LIN {X 0,Y 303.722,Z 314.6,A -85,B 0,C 180,E1 -15936.643,E2 -15936.643} C_VEL
LIN {X 0,Y 304.019,Z 311.814,A -85,B 0,C 180,E1 -15938.642,E2 -15938.642} C_VEL
LIN {X 0,Y 304.561,Z 308.03,A -85,B 0,C 180,E1 -15940.638,E2 -15940.638} C_VEL
LIN {X 0,Y 305.432,Z 303.153,A -85,B 0,C 180,E1 -15942.626,E2 -15942.626} C_VEL
LIN {X 0,Y 306.814,Z 297.041,A -85,B 0,C 180,E1 -15944.594,E2 -15944.594} C_VEL
LIN {X 0,Y 308.414,Z 289.012,A -85,B 0,C 180,E1 -15946.664,E2 -15946.664} C_VEL
LIN {X 0,Y 310.224,Z 280.048,A -85,B 0,C 180,E1 -15948.491,E2 -15948.491} C_VEL
LIN {X 0,Y 312.464,Z 269.264,A -85,B 0,C 180,E1 -15950.231,E2 -15950.231} C_VEL
LIN {X 0,Y 314.317,Z 259.561,A -85,B 0,C 180,E1 -15951.477,E2 -15951.477} C_VEL
LIN {X 0,Y 316.058,Z 249.097,A -85,B 0,C 180,E1 -15952.555,E2 -15952.555} C_VEL
LIN {X 0,Y 317.837,Z 236.54,A -85,B 0,C 180,E1 -15953.54,E2 -15953.54} C_VEL
LIN {X 0,Y 319.26,Z 224.054,A -85,B 0,C 180,E1 -15954.247,E2 -15954.247} C_VEL
LIN {X 0,Y 320.237,Z 211.153,A -85,B 0,C 180,E1 -15954.73,E2 -15954.73} C_VEL
LIN {X 0,Y 321.791,Z 150.859,A -85,B 0,C 180,E1 -15956.133,E2 -15956.133} C_VEL
LIN {X 0,Y 318.654,Z 131.101,A -85,B 0,C 180,E1 -15956.979,E2 -15956.979} C_VEL
LIN {X 0,Y 314.024,Z 108.711,A -85,B 0,C 180,E1 -15958.092,E2 -15958.092} C_VEL
LIN {X 0,Y 312.285,Z 103.067,A -85,B 0,C 180,E1 -15958.447,E2 -15958.447} C_VEL
LIN {X 0,Y 310.254,Z 93.46,A -85,B 0,C 180,E1 -15961.399,E2 -15961.399} C_VEL
LIN {X 0,Y 308.062,Z 84.289,A -85,B 0,C 180,E1 -15964.395,E2 -15964.395} C_VEL
LIN {X 0,Y 305.495,Z 74.434,A -85,B 0,C 180,E1 -15967.849,E2 -15967.849} C_VEL
LIN {X 0,Y 305.439,Z 74.437,A -85,B 0,C 180,E1 -15971.856,E2 -15971.856} C_VEL
LIN {X 0,Y 305.408,Z 74.423,A -85,B 0,C 180,E1 -15975.509,E2 -15975.509} C_VEL
LIN {X 0,Y 305.473,Z 74.434,A -85,B 0,C 180,E1 -15978.149,E2 -15978.149} C_VEL
LIN {X 0,Y 305.506,Z 74.426,A -85,B 0,C 180,E1 -15981.602,E2 -15981.602} C_VEL
LIN {X 0,Y 305.46,Z 74.433,A -85,B 0,C 180,E1 -15984.887,E2 -15984.887} C_VEL
LIN {X 0,Y 305.45,Z 74.435,A -85,B 0,C 180,E1 -15988.354,E2 -15988.354} C_VEL
LIN {X 0,Y 305.518,Z 74.43,A -85,B 0,C 180,E1 -15991.114,E2 -15991.114} C_VEL
LIN {X 0,Y 305.569,Z 74.416,A -85,B 0,C 180,E1 -15994.088,E2 -15994.088} C_VEL
LIN {X 0,Y 305.501,Z 74.421,A -85,B 0,C 180,E1 -15998.403,E2 -15998.403} C_VEL
LIN {X 0,Y 305.589,Z 74.412,A -85,B 0,C 180,E1 -16001.218,E2 -16001.218} C_VEL
LIN {X 0,Y 305.646,Z 74.411,A -85,B 0,C 180,E1 -16005.349,E2 -16005.349} C_VEL
LIN {X 0,Y 305.636,Z 74.412,A -85,B 0,C 180,E1 -16009.4,E2 -16009.4} C_VEL
LIN {X 0,Y 305.805,Z 74.381,A -85,B 0,C 180,E1 -16012.074,E2 -16012.074} C_VEL
LIN {X 0,Y 305.684,Z 74.407,A -85,B 0,C 180,E1 -16014.724,E2 -16014.724} C_VEL
LIN {X 0,Y 305.955,Z 74.368,A -85,B 0,C 180,E1 -16018.684,E2 -16018.684} C_VEL
LIN {X 0,Y 305.953,Z 74.372,A -85,B 0,C 180,E1 -16021.317,E2 -16021.317} C_VEL
LIN {X 0,Y 305.68,Z 74.409,A -85,B 0,C 180,E1 -16025.277,E2 -16025.277} C_VEL
LIN {X 0,Y 305.769,Z 74.384,A -85,B 0,C 180,E1 -16027.927,E2 -16027.927} C_VEL
LIN {X 0,Y 305.597,Z 74.412,A -85,B 0,C 180,E1 -16031.946,E2 -16031.946} C_VEL
LIN {X 0,Y 305.607,Z 74.418,A -85,B 0,C 180,E1 -16035.015,E2 -16035.015} C_VEL
LIN {X 0,Y 305.542,Z 74.426,A -85,B 0,C 180,E1 -16039.428,E2 -16039.428} C_VEL
LIN {X 0,Y 305.484,Z 74.43,A -85,B 0,C 180,E1 -16043.04,E2 -16043.04} C_VEL
LIN {X 0,Y 305.476,Z 74.426,A -85,B 0,C 180,E1 -16046.201,E2 -16046.201} C_VEL
LIN {X 0,Y 305.461,Z 74.429,A -85,B 0,C 180,E1 -16049.039,E2 -16049.039} C_VEL
LIN {X 0,Y 305.436,Z 74.436,A -85,B 0,C 180,E1 -16051.954,E2 -16051.954} C_VEL
LIN {X 0,Y 305.461,Z 74.43,A -85,B 0,C 180,E1 -16055.114,E2 -16055.114} C_VEL
LIN {X 0,Y 305.434,Z 74.442,A -85,B 0,C 180,E1 -16058.526,E2 -16058.526} C_VEL
LIN {X 0,Y 305.426,Z 74.431,A -85,B 0,C 180,E1 -16061.86,E2 -16061.86} C_VEL
LIN {X 0,Y 305.411,Z 74.441,A -85,B 0,C 180,E1 -16065.938,E2 -16065.938} C_VEL
LIN {X 0,Y 305.48,Z 74.708,A -85,B 0,C 180,E1 -16066.355,E2 -16066.355} C_VEL
LIN {X 0,Y 305.822,Z 75.973,A -85,B 0,C 180,E1 -16066.792,E2 -16066.792} C_VEL
LIN {X 0,Y 313.965,Z 91.34,A -85,B 0,C 180,E1 -16068.219,E2 -16068.219} C_VEL
LIN {X 0,Y 321.333,Z 106.833,A -85,B 0,C 180,E1 -16069.468,E2 -16069.468} C_VEL
LIN {X 0,Y 323.152,Z 111.258,A -85,B 0,C 180,E1 -16069.78,E2 -16069.78} C_VEL
LIN {X 0,Y 320.986,Z 181.678,A -85,B 0,C 180,E1 -16071.391,E2 -16071.391} C_VEL
LIN {X 0,Y 320.123,Z 194.669,A -85,B 0,C 180,E1 -16071.92,E2 -16071.92} C_VEL
LIN {X 0,Y 319.072,Z 207.723,A -85,B 0,C 180,E1 -16072.738,E2 -16072.738} C_VEL
LIN {X 0,Y 317.642,Z 219.301,A -85,B 0,C 180,E1 -16073.712,E2 -16073.712} C_VEL
LIN {X 0,Y 315.904,Z 230.916,A -85,B 0,C 180,E1 -16074.989,E2 -16074.989} C_VEL
LIN {X 0,Y 314.114,Z 240.957,A -85,B 0,C 180,E1 -16076.375,E2 -16076.375} C_VEL
LIN {X 0,Y 312.149,Z 250.688,A -85,B 0,C 180,E1 -16078.056,E2 -16078.056} C_VEL
LIN {X 0,Y 310.584,Z 258.046,A -85,B 0,C 180,E1 -16079.627,E2 -16079.627} C_VEL
LIN {X 0,Y 308.977,Z 265.076,A -85,B 0,C 180,E1 -16081.468,E2 -16081.468} C_VEL
LIN {X 0,Y 307.432,Z 271.447,A -85,B 0,C 180,E1 -16083.564,E2 -16083.564} C_VEL
LIN {X 0,Y 306.27,Z 276.256,A -85,B 0,C 180,E1 -16085.604,E2 -16085.604} C_VEL
LIN {X 0,Y 305.351,Z 279.946,A -85,B 0,C 180,E1 -16087.681,E2 -16087.681} C_VEL
LIN {X 0,Y 304.641,Z 282.538,A -85,B 0,C 180,E1 -16089.755,E2 -16089.755} C_VEL
LIN {X 0,Y 304.213,Z 283.817,A -85,B 0,C 180,E1 -16091.298,E2 -16091.298} C_VEL
LIN {X 0,Y 303.812,Z 284.734,A -85,B 0,C 180,E1 -16093.884,E2 -16093.884} C_VEL
LIN {X 0,Y 303.721,Z 284.241,A -85,B 0,C 180,E1 -16096.379,E2 -16096.379} C_VEL
LIN {X 0,Y 303.759,Z 283.153,A -85,B 0,C 180,E1 -16097.982,E2 -16097.982} C_VEL
LIN {X 0,Y 303.804,Z 281.805,A -85,B 0,C 180,E1 -16099.335,E2 -16099.335} C_VEL
LIN {X 0,Y 304.108,Z 278.947,A -85,B 0,C 180,E1 -16101.361,E2 -16101.361} C_VEL
LIN {X 0,Y 304.502,Z 275.058,A -85,B 0,C 180,E1 -16103.374,E2 -16103.374} C_VEL
LIN {X 0,Y 304.981,Z 270.045,A -85,B 0,C 180,E1 -16105.374,E2 -16105.374} C_VEL
LIN {X 0,Y 305.676,Z 263.747,A -85,B 0,C 180,E1 -16107.365,E2 -16107.365} C_VEL
LIN {X 0,Y 306.671,Z 255.843,A -85,B 0,C 180,E1 -16109.344,E2 -16109.344} C_VEL
LIN {X 0,Y 307.685,Z 247.786,A -85,B 0,C 180,E1 -16110.982,E2 -16110.982} C_VEL
LIN {X 0,Y 308.861,Z 237.964,A -85,B 0,C 180,E1 -16112.609,E2 -16112.609} C_VEL
LIN {X 0,Y 310.052,Z 227.133,A -85,B 0,C 180,E1 -16114.044,E2 -16114.044} C_VEL
LIN {X 0,Y 311.02,Z 216.232,A -85,B 0,C 180,E1 -16115.186,E2 -16115.186} C_VEL
LIN {X 0,Y 311.857,Z 204.447,A -85,B 0,C 180,E1 -16116.146,E2 -16116.146} C_VEL
LIN {X 0,Y 312.535,Z 191.764,A -85,B 0,C 180,E1 -16116.902,E2 -16116.902} C_VEL
LIN {X 0,Y 313.021,Z 179.469,A -85,B 0,C 180,E1 -16117.378,E2 -16117.378} C_VEL
LIN {X 0,Y 314.626,Z 100.764,A -85,B 0,C 180,E1 -16119.182,E2 -16119.182} C_VEL
LIN {X 0,Y 309.281,Z 84.113,A -85,B 0,C 180,E1 -16119.931,E2 -16119.931} C_VEL
LIN {X 0,Y 305.662,Z 74.413,A -85,B 0,C 180,E1 -16120.435,E2 -16120.435} C_VEL
LIN {X 0,Y 305.643,Z 74.414,A -85,B 0,C 180,E1 -16125.035,E2 -16125.035} C_VEL
LIN {X 0,Y 305.58,Z 74.418,A -85,B 0,C 180,E1 -16129.445,E2 -16129.445} C_VEL
LIN {X 0,Y 305.49,Z 74.428,A -85,B 0,C 180,E1 -16133.039,E2 -16133.039} C_VEL
LIN {X 0,Y 305.536,Z 74.425,A -85,B 0,C 180,E1 -16136.221,E2 -16136.221} C_VEL
LIN {X 0,Y 305.492,Z 74.428,A -85,B 0,C 180,E1 -16139.047,E2 -16139.047} C_VEL
LIN {X 0,Y 305.447,Z 74.436,A -85,B 0,C 180,E1 -16141.952,E2 -16141.952} C_VEL
LIN {X 0,Y 305.467,Z 74.43,A -85,B 0,C 180,E1 -16145.113,E2 -16145.113} C_VEL
LIN {X 0,Y 305.472,Z 74.431,A -85,B 0,C 180,E1 -16148.533,E2 -16148.533} C_VEL
LIN {X 0,Y 305.481,Z 74.43,A -85,B 0,C 180,E1 -16152.59,E2 -16152.59} C_VEL
LIN {X 0,Y 305.447,Z 74.434,A -85,B 0,C 180,E1 -16156.348,E2 -16156.348} C_VEL
LIN {X 0,Y 305.449,Z 74.432,A -85,B 0,C 180,E1 -16160.05,E2 -16160.05} C_VEL
LIN {X 0,Y 304.746,Z 74.522,A -85,B 0,C 180,E1 -16161.151,E2 -16161.151} C_VEL
LIN {X 0,Y 301.917,Z 74.87,A -85,B 0,C 180,E1 -16162.945,E2 -16162.945} C_VEL
LIN {X 0,Y 299.531,Z 75.166,A -85,B 0,C 180,E1 -16164.4,E2 -16164.4} C_VEL
LIN {X 0,Y 298.487,Z 75.294,A -85,B 0,C 180,E1 -16165.525,E2 -16165.525} C_VEL
LIN {X 0,Y 298.39,Z 75.305,A -85,B 0,C 180,E1 -16165.907,E2 -16165.907} C_VEL
LIN {X 0,Y 298.395,Z 75.314,A -85,B 0,C 180,E1 -16168.791,E2 -16168.791} C_VEL
LIN {X 0,Y 298.46,Z 75.305,A -85,B 0,C 180,E1 -16171.903,E2 -16171.903} C_VEL
LIN {X 0,Y 298.486,Z 75.301,A -85,B 0,C 180,E1 -16174.924,E2 -16174.924} C_VEL
LIN {X 0,Y 298.454,Z 75.306,A -85,B 0,C 180,E1 -16179.315,E2 -16179.315} C_VEL
LIN {X 0,Y 298.541,Z 75.297,A -85,B 0,C 180,E1 -16182.179,E2 -16182.179} C_VEL
LIN {X 0,Y 298.596,Z 75.287,A -85,B 0,C 180,E1 -16184.995,E2 -16184.995} C_VEL
LIN {X 0,Y 298.594,Z 75.288,A -85,B 0,C 180,E1 -16189.146,E2 -16189.146} C_VEL
LIN {X 0,Y 298.744,Z 75.27,A -85,B 0,C 180,E1 -16191.885,E2 -16191.885} C_VEL
LIN {X 0,Y 298.658,Z 75.28,A -85,B 0,C 180,E1 -16194.599,E2 -16194.599} C_VEL
LIN {X 0,Y 298.924,Z 75.245,A -85,B 0,C 180,E1 -16198.652,E2 -16198.652} C_VEL
LIN {X 0,Y 298.924,Z 75.246,A -85,B 0,C 180,E1 -16201.347,E2 -16201.347} C_VEL
LIN {X 0,Y 298.778,Z 75.264,A -85,B 0,C 180,E1 -16206.754,E2 -16206.754} C_VEL
LIN {X 0,Y 298.628,Z 75.287,A -85,B 0,C 180,E1 -16209.482,E2 -16209.482} C_VEL
LIN {X 0,Y 298.555,Z 75.294,A -85,B 0,C 180,E1 -16213.615,E2 -16213.615} C_VEL
LIN {X 0,Y 298.551,Z 75.292,A -85,B 0,C 180,E1 -16216.408,E2 -16216.408} C_VEL
LIN {X 0,Y 298.512,Z 75.299,A -85,B 0,C 180,E1 -16219.653,E2 -16219.653} C_VEL
LIN {X 0,Y 298.43,Z 75.309,A -85,B 0,C 180,E1 -16223.6,E2 -16223.6} C_VEL
LIN {X 0,Y 298.487,Z 75.303,A -85,B 0,C 180,E1 -16226.574,E2 -16226.574} C_VEL
LIN {X 0,Y 298.423,Z 75.307,A -85,B 0,C 180,E1 -16229.641,E2 -16229.641} C_VEL
LIN {X 0,Y 298.397,Z 75.316,A -85,B 0,C 180,E1 -16232.8,E2 -16232.8} C_VEL
LIN {X 0,Y 298.448,Z 75.309,A -85,B 0,C 180,E1 -16236.807,E2 -16236.807} C_VEL
LIN {X 0,Y 298.388,Z 75.315,A -85,B 0,C 180,E1 -16241.087,E2 -16241.087} C_VEL
LIN {X 0,Y 298.4,Z 75.312,A -85,B 0,C 180,E1 -16243.103,E2 -16243.103} C_VEL
LIN {X 0,Y 298.404,Z 75.313,A -85,B 0,C 180,E1 -16246.92,E2 -16246.92} C_VEL
LIN {X 0,Y 298.416,Z 75.312,A -85,B 0,C 180,E1 -16251.003,E2 -16251.003} C_VEL
LIN {X 0,Y 298.433,Z 75.314,A -85,B 0,C 180,E1 -16253.932,E2 -16253.932} C_VEL
LIN {X 0,Y 298.456,Z 75.334,A -85,B 0,C 180,E1 -16257.363,E2 -16257.363} C_VEL
LIN {X 0,Y 301.125,Z 88.007,A -85,B 0,C 180,E1 -16261.034,E2 -16261.034} C_VEL
LIN {X 0,Y 302.351,Z 95.258,A -85,B 0,C 180,E1 -16263.046,E2 -16263.046} C_VEL
LIN {X 0,Y 301.429,Z 103.913,A -85,B 0,C 180,E1 -16265.263,E2 -16265.263} C_VEL
LIN {X 0,Y 306.811,Z 147.996,A -85,B 0,C 180,E1 -16266.715,E2 -16266.715} C_VEL
LIN {X 0,Y 306.88,Z 159.405,A -85,B 0,C 180,E1 -16266.998,E2 -16266.998} C_VEL
LIN {X 0,Y 305.694,Z 213.727,A -85,B 0,C 180,E1 -16268.296,E2 -16268.296} C_VEL
LIN {X 0,Y 304.904,Z 227.31,A -85,B 0,C 180,E1 -16268.89,E2 -16268.89} C_VEL
LIN {X 0,Y 303.903,Z 239.769,A -85,B 0,C 180,E1 -16269.702,E2 -16269.702} C_VEL
LIN {X 0,Y 302.735,Z 250.891,A -85,B 0,C 180,E1 -16270.681,E2 -16270.681} C_VEL
LIN {X 0,Y 301.478,Z 261.198,A -85,B 0,C 180,E1 -16271.832,E2 -16271.832} C_VEL
LIN {X 0,Y 300.34,Z 271.925,A -85,B 0,C 180,E1 -16273.342,E2 -16273.342} C_VEL
LIN {X 0,Y 299.397,Z 280.34,A -85,B 0,C 180,E1 -16274.797,E2 -16274.797} C_VEL
LIN {X 0,Y 298.329,Z 289.451,A -85,B 0,C 180,E1 -16276.721,E2 -16276.721} C_VEL
LIN {X 0,Y 297.404,Z 297.125,A -85,B 0,C 180,E1 -16278.757,E2 -16278.757} C_VEL
LIN {X 0,Y 296.926,Z 304.228,A -85,B 0,C 180,E1 -16281.149,E2 -16281.149} C_VEL
LIN {X 0,Y 296.685,Z 308.907,A -85,B 0,C 180,E1 -16283.197,E2 -16283.197} C_VEL
LIN {X 0,Y 296.635,Z 312.451,A -85,B 0,C 180,E1 -16285.243,E2 -16285.243} C_VEL
LIN {X 0,Y 296.692,Z 314.96,A -85,B 0,C 180,E1 -16287.284,E2 -16287.284} C_VEL
LIN {X 0,Y 296.771,Z 316.11,A -85,B 0,C 180,E1 -16288.643,E2 -16288.643} C_VEL
LIN {X 0,Y 296.857,Z 316.815,A -85,B 0,C 180,E1 -16290,E2 -16290} C_VEL
LIN {X 0,Y 296.623,Z 317.027,A -85,B 0,C 180,E1 -16292.716,E2 -16292.716} C_VEL
LIN {X 0,Y 296.596,Z 316.546,A -85,B 0,C 180,E1 -16294.076,E2 -16294.076} C_VEL
LIN {X 0,Y 296.644,Z 314.324,A -85,B 0,C 180,E1 -16296.803,E2 -16296.803} C_VEL
LIN {X 0,Y 296.975,Z 311.593,A -85,B 0,C 180,E1 -16298.848,E2 -16298.848} C_VEL
LIN {X 0,Y 297.544,Z 307.864,A -85,B 0,C 180,E1 -16300.892,E2 -16300.892} C_VEL
LIN {X 0,Y 298.487,Z 303.048,A -85,B 0,C 180,E1 -16302.925,E2 -16302.925} C_VEL
LIN {X 0,Y 300.18,Z 295.88,A -85,B 0,C 180,E1 -16305.271,E2 -16305.271} C_VEL
LIN {X 0,Y 301.737,Z 288.176,A -85,B 0,C 180,E1 -16307.261,E2 -16307.261} C_VEL
LIN {X 0,Y 303.918,Z 278.435,A -85,B 0,C 180,E1 -16309.239,E2 -16309.239} C_VEL
LIN {X 0,Y 306.043,Z 268.475,A -85,B 0,C 180,E1 -16310.851,E2 -16310.851} C_VEL
LIN {X 0,Y 308.045,Z 258.665,A -85,B 0,C 180,E1 -16312.113,E2 -16312.113} C_VEL
LIN {X 0,Y 309.834,Z 248.056,A -85,B 0,C 180,E1 -16313.21,E2 -16313.21} C_VEL
LIN {X 0,Y 311.716,Z 235.322,A -85,B 0,C 180,E1 -16314.208,E2 -16314.208} C_VEL
LIN {X 0,Y 313.192,Z 222.536,A -85,B 0,C 180,E1 -16314.926,E2 -16314.926} C_VEL
LIN {X 0,Y 314.069,Z 209.411,A -85,B 0,C 180,E1 -16315.405,E2 -16315.405} C_VEL
LIN {X 0,Y 315.77,Z 152.738,A -85,B 0,C 180,E1 -16316.726,E2 -16316.726} C_VEL
LIN {X 0,Y 312.775,Z 133.284,A -85,B 0,C 180,E1 -16317.577,E2 -16317.577} C_VEL
LIN {X 0,Y 308.218,Z 110.954,A -85,B 0,C 180,E1 -16318.718,E2 -16318.718} C_VEL
LIN {X 0,Y 306.786,Z 106.516,A -85,B 0,C 180,E1 -16319.016,E2 -16319.016} C_VEL
LIN {X 0,Y 305.043,Z 102.497,A -85,B 0,C 180,E1 -16319.37,E2 -16319.37} C_VEL
LIN {X 0,Y 302.639,Z 91.519,A -85,B 0,C 180,E1 -16322.9,E2 -16322.9} C_VEL
LIN {X 0,Y 299.836,Z 80.463,A -85,B 0,C 180,E1 -16326.743,E2 -16326.743} C_VEL
LIN {X 0,Y 298.421,Z 75.312,A -85,B 0,C 180,E1 -16328.681,E2 -16328.681} C_VEL
LIN {X 0,Y 298.397,Z 75.317,A -85,B 0,C 180,E1 -16333.103,E2 -16333.103} C_VEL
LIN {X 0,Y 298.43,Z 75.302,A -85,B 0,C 180,E1 -16336.926,E2 -16336.926} C_VEL
LIN {X 0,Y 298.424,Z 75.313,A -85,B 0,C 180,E1 -16341.001,E2 -16341.001} C_VEL
LIN {X 0,Y 298.43,Z 75.311,A -85,B 0,C 180,E1 -16343.932,E2 -16343.932} C_VEL
LIN {X 0,Y 298.393,Z 75.315,A -85,B 0,C 180,E1 -16347.983,E2 -16347.983} C_VEL
LIN {X 0,Y 298.461,Z 75.306,A -85,B 0,C 180,E1 -16351.904,E2 -16351.904} C_VEL
LIN {X 0,Y 298.483,Z 75.305,A -85,B 0,C 180,E1 -16354.924,E2 -16354.924} C_VEL
LIN {X 0,Y 298.454,Z 75.307,A -85,B 0,C 180,E1 -16359.316,E2 -16359.316} C_VEL
LIN {X 0,Y 298.536,Z 75.286,A -85,B 0,C 180,E1 -16362.179,E2 -16362.179} C_VEL
LIN {X 0,Y 298.591,Z 75.29,A -85,B 0,C 180,E1 -16364.995,E2 -16364.995} C_VEL
LIN {X 0,Y 298.591,Z 75.29,A -85,B 0,C 180,E1 -16369.147,E2 -16369.147} C_VEL
LIN {X 0,Y 298.752,Z 75.26,A -85,B 0,C 180,E1 -16371.886,E2 -16371.886} C_VEL
LIN {X 0,Y 298.655,Z 75.283,A -85,B 0,C 180,E1 -16374.599,E2 -16374.599} C_VEL
LIN {X 0,Y 298.921,Z 75.243,A -85,B 0,C 180,E1 -16378.653,E2 -16378.653} C_VEL
LIN {X 0,Y 298.919,Z 75.247,A -85,B 0,C 180,E1 -16381.348,E2 -16381.348} C_VEL
LIN {X 0,Y 298.773,Z 75.265,A -85,B 0,C 180,E1 -16386.755,E2 -16386.755} C_VEL
LIN {X 0,Y 298.623,Z 75.282,A -85,B 0,C 180,E1 -16389.483,E2 -16389.483} C_VEL
LIN {X 0,Y 298.543,Z 75.288,A -85,B 0,C 180,E1 -16393.616,E2 -16393.616} C_VEL
LIN {X 0,Y 298.485,Z 75.302,A -85,B 0,C 180,E1 -16396.413,E2 -16396.413} C_VEL
LIN {X 0,Y 298.482,Z 75.305,A -85,B 0,C 180,E1 -16399.64,E2 -16399.64} C_VEL
LIN {X 0,Y 298.423,Z 75.312,A -85,B 0,C 180,E1 -16403.601,E2 -16403.601} C_VEL
LIN {X 0,Y 298.415,Z 75.308,A -85,B 0,C 180,E1 -16406.582,E2 -16406.582} C_VEL
LIN {X 0,Y 298.399,Z 75.309,A -85,B 0,C 180,E1 -16409.644,E2 -16409.644} C_VEL
LIN {X 0,Y 298.392,Z 75.312,A -85,B 0,C 180,E1 -16412.801,E2 -16412.801} C_VEL
LIN {X 0,Y 298.441,Z 75.312,A -85,B 0,C 180,E1 -16416.807,E2 -16416.807} C_VEL
LIN {X 0,Y 298.38,Z 75.306,A -85,B 0,C 180,E1 -16421.087,E2 -16421.087} C_VEL
LIN {X 0,Y 298.399,Z 75.324,A -85,B 0,C 180,E1 -16423.104,E2 -16423.104} C_VEL
LIN {X 0,Y 298.375,Z 75.401,A -85,B 0,C 180,E1 -16425.5,E2 -16425.5} C_VEL
LIN {X 0,Y 298.533,Z 76.217,A -85,B 0,C 180,E1 -16425.831,E2 -16425.831} C_VEL
LIN {X 0,Y 300.086,Z 79.172,A -85,B 0,C 180,E1 -16426.129,E2 -16426.129} C_VEL
LIN {X 0,Y 307.562,Z 92.858,A -85,B 0,C 180,E1 -16427.486,E2 -16427.486} C_VEL
LIN {X 0,Y 315.028,Z 108.392,A -85,B 0,C 180,E1 -16428.8,E2 -16428.8} C_VEL
LIN {X 0,Y 317.041,Z 113.075,A -85,B 0,C 180,E1 -16429.154,E2 -16429.154} C_VEL
LIN {X 0,Y 314.826,Z 182.102,A -85,B 0,C 180,E1 -16430.762,E2 -16430.762} C_VEL
LIN {X 0,Y 313.876,Z 195.801,A -85,B 0,C 180,E1 -16431.338,E2 -16431.338} C_VEL
LIN {X 0,Y 312.81,Z 208.298,A -85,B 0,C 180,E1 -16432.144,E2 -16432.144} C_VEL
LIN {X 0,Y 311.415,Z 219.156,A -85,B 0,C 180,E1 -16433.068,E2 -16433.068} C_VEL
LIN {X 0,Y 309.73,Z 229.943,A -85,B 0,C 180,E1 -16434.249,E2 -16434.249} C_VEL
LIN {X 0,Y 307.726,Z 240.977,A -85,B 0,C 180,E1 -16435.779,E2 -16435.779} C_VEL
LIN {X 0,Y 305.818,Z 249.892,A -85,B 0,C 180,E1 -16437.313,E2 -16437.313} C_VEL
LIN {X 0,Y 303.966,Z 258.346,A -85,B 0,C 180,E1 -16439.128,E2 -16439.128} C_VEL
LIN {X 0,Y 302.147,Z 265.846,A -85,B 0,C 180,E1 -16441.142,E2 -16441.142} C_VEL
LIN {X 0,Y 300.677,Z 271.54,A -85,B 0,C 180,E1 -16443.055,E2 -16443.055} C_VEL
LIN {X 0,Y 299.487,Z 276.156,A -85,B 0,C 180,E1 -16445.014,E2 -16445.014} C_VEL
LIN {X 0,Y 298.725,Z 279.091,A -85,B 0,C 180,E1 -16446.57,E2 -16446.57} C_VEL
LIN {X 0,Y 298.212,Z 281.006,A -85,B 0,C 180,E1 -16447.848,E2 -16447.848} C_VEL
LIN {X 0,Y 297.714,Z 282.682,A -85,B 0,C 180,E1 -16449.262,E2 -16449.262} C_VEL
LIN {X 0,Y 297.201,Z 284.199,A -85,B 0,C 180,E1 -16451.068,E2 -16451.068} C_VEL
LIN {X 0,Y 296.761,Z 285.1,A -85,B 0,C 180,E1 -16453.49,E2 -16453.49} C_VEL
LIN {X 0,Y 296.635,Z 284.634,A -85,B 0,C 180,E1 -16456.264,E2 -16456.264} C_VEL
LIN {X 0,Y 296.651,Z 283.735,A -85,B 0,C 180,E1 -16457.689,E2 -16457.689} C_VEL
LIN {X 0,Y 296.691,Z 282.44,A -85,B 0,C 180,E1 -16459.077,E2 -16459.077} C_VEL
LIN {X 0,Y 296.982,Z 279.693,A -85,B 0,C 180,E1 -16461.152,E2 -16461.152} C_VEL
LIN {X 0,Y 297.391,Z 275.921,A -85,B 0,C 180,E1 -16463.215,E2 -16463.215} C_VEL
LIN {X 0,Y 297.857,Z 271.035,A -85,B 0,C 180,E1 -16465.263,E2 -16465.263} C_VEL
LIN {X 0,Y 298.564,Z 264.877,A -85,B 0,C 180,E1 -16467.302,E2 -16467.302} C_VEL
LIN {X 0,Y 299.561,Z 257.21,A -85,B 0,C 180,E1 -16469.328,E2 -16469.328} C_VEL
LIN {X 0,Y 300.582,Z 249.354,A -85,B 0,C 180,E1 -16471.005,E2 -16471.005} C_VEL
LIN {X 0,Y 301.764,Z 239.77,A -85,B 0,C 180,E1 -16472.67,E2 -16472.67} C_VEL
LIN {X 0,Y 303.023,Z 228.766,A -85,B 0,C 180,E1 -16474.204,E2 -16474.204} C_VEL
LIN {X 0,Y 304.13,Z 217.193,A -85,B 0,C 180,E1 -16475.47,E2 -16475.47} C_VEL
LIN {X 0,Y 305.065,Z 204.451,A -85,B 0,C 180,E1 -16476.532,E2 -16476.532} C_VEL
LIN {X 0,Y 305.773,Z 191.588,A -85,B 0,C 180,E1 -16477.304,E2 -16477.304} C_VEL
LIN {X 0,Y 306.27,Z 178.865,A -85,B 0,C 180,E1 -16477.79,E2 -16477.79} C_VEL
LIN {X 0,Y 307.887,Z 101.929,A -85,B 0,C 180,E1 -16479.587,E2 -16479.587} C_VEL
LIN {X 0,Y 302.49,Z 85.456,A -85,B 0,C 180,E1 -16480.359,E2 -16480.359} C_VEL
LIN {X 0,Y 298.69,Z 75.916,A -85,B 0,C 180,E1 -16480.869,E2 -16480.869} C_VEL
LIN {X 0,Y 298.577,Z 75.296,A -85,B 0,C 180,E1 -16480.94,E2 -16480.94} C_VEL
LIN {X 0,Y 298.61,Z 75.29,A -85,B 0,C 180,E1 -16485.209,E2 -16485.209} C_VEL
LIN {X 0,Y 298.543,Z 75.294,A -85,B 0,C 180,E1 -16489.243,E2 -16489.243} C_VEL
LIN {X 0,Y 298.433,Z 75.309,A -85,B 0,C 180,E1 -16493.6,E2 -16493.6} C_VEL
LIN {X 0,Y 298.491,Z 75.3,A -85,B 0,C 180,E1 -16496.575,E2 -16496.575} C_VEL
LIN {X 0,Y 298.421,Z 75.312,A -85,B 0,C 180,E1 -16499.641,E2 -16499.641} C_VEL
LIN {X 0,Y 298.4,Z 75.31,A -85,B 0,C 180,E1 -16502.8,E2 -16502.8} C_VEL
LIN {X 0,Y 298.469,Z 75.304,A -85,B 0,C 180,E1 -16506.812,E2 -16506.812} C_VEL
LIN {X 0,Y 298.416,Z 75.311,A -85,B 0,C 180,E1 -16511.093,E2 -16511.093} C_VEL
LIN {X 0,Y 298.43,Z 75.311,A -85,B 0,C 180,E1 -16513.109,E2 -16513.109} C_VEL
LIN {X 0,Y 298.406,Z 75.312,A -85,B 0,C 180,E1 -16516.921,E2 -16516.921} C_VEL
LIN {X 0,Y 298.402,Z 75.313,A -85,B 0,C 180,E1 -16521.007,E2 -16521.007} C_VEL
LIN {X 0,Y 298.421,Z 75.298,A -85,B 0,C 180,E1 -16523.93,E2 -16523.93} C_VEL
LIN {X 0,Y 298.39,Z 75.305,A -85,B 0,C 180,E1 -16525.907,E2 -16525.907} C_VEL
LIN {X 0,Y 297.689,Z 75.398,A -85,B 0,C 180,E1 -16527.034,E2 -16527.034} C_VEL
LIN {X 0,Y 294.834,Z 75.758,A -85,B 0,C 180,E1 -16528.869,E2 -16528.869} C_VEL
LIN {X 0,Y 292.448,Z 76.055,A -85,B 0,C 180,E1 -16530.359,E2 -16530.359} C_VEL
LIN {X 0,Y 291.445,Z 76.18,A -85,B 0,C 180,E1 -16531.513,E2 -16531.513} C_VEL
LIN {X 0,Y 291.373,Z 76.188,A -85,B 0,C 180,E1 -16531.903,E2 -16531.903} C_VEL
LIN {X 0,Y 291.416,Z 76.183,A -85,B 0,C 180,E1 -16534.271,E2 -16534.271} C_VEL
LIN {X 0,Y 291.385,Z 76.186,A -85,B 0,C 180,E1 -16537.299,E2 -16537.299} C_VEL
LIN {X 0,Y 291.461,Z 76.18,A -85,B 0,C 180,E1 -16540.27,E2 -16540.27} C_VEL
LIN {X 0,Y 291.558,Z 76.165,A -85,B 0,C 180,E1 -16544.623,E2 -16544.623} C_VEL
LIN {X 0,Y 291.538,Z 76.167,A -85,B 0,C 180,E1 -16548.88,E2 -16548.88} C_VEL
LIN {X 0,Y 291.691,Z 76.147,A -85,B 0,C 180,E1 -16551.688,E2 -16551.688} C_VEL
LIN {X 0,Y 291.629,Z 76.157,A -85,B 0,C 180,E1 -16554.468,E2 -16554.468} C_VEL
LIN {X 0,Y 291.891,Z 76.121,A -85,B 0,C 180,E1 -16558.62,E2 -16558.62} C_VEL
LIN {X 0,Y 291.891,Z 76.122,A -85,B 0,C 180,E1 -16561.379,E2 -16561.379} C_VEL
LIN {X 0,Y 291.725,Z 76.143,A -85,B 0,C 180,E1 -16566.918,E2 -16566.918} C_VEL
LIN {X 0,Y 291.57,Z 76.165,A -85,B 0,C 180,E1 -16569.714,E2 -16569.714} C_VEL
LIN {X 0,Y 291.524,Z 76.168,A -85,B 0,C 180,E1 -16573.95,E2 -16573.95} C_VEL
LIN {X 0,Y 291.489,Z 76.173,A -85,B 0,C 180,E1 -16576.817,E2 -16576.817} C_VEL
LIN {X 0,Y 291.453,Z 76.178,A -85,B 0,C 180,E1 -16579.874,E2 -16579.874} C_VEL
LIN {X 0,Y 291.384,Z 76.187,A -85,B 0,C 180,E1 -16584.207,E2 -16584.207} C_VEL
LIN {X 0,Y 291.422,Z 76.183,A -85,B 0,C 180,E1 -16587.271,E2 -16587.271} C_VEL
LIN {X 0,Y 291.339,Z 76.192,A -85,B 0,C 180,E1 -16590.436,E2 -16590.436} C_VEL
LIN {X 0,Y 291.347,Z 76.191,A -85,B 0,C 180,E1 -16593.698,E2 -16593.698} C_VEL
LIN {X 0,Y 291.377,Z 76.188,A -85,B 0,C 180,E1 -16597.254,E2 -16597.254} C_VEL
LIN {X 0,Y 291.334,Z 76.196,A -85,B 0,C 180,E1 -16600.642,E2 -16600.642} C_VEL
LIN {X 0,Y 291.292,Z 76.197,A -85,B 0,C 180,E1 -16604.402,E2 -16604.402} C_VEL
LIN {X 0,Y 291.328,Z 76.197,A -85,B 0,C 180,E1 -16608.404,E2 -16608.404} C_VEL
LIN {X 0,Y 291.366,Z 76.191,A -85,B 0,C 180,E1 -16611.16,E2 -16611.16} C_VEL
LIN {X 0,Y 291.387,Z 76.189,A -85,B 0,C 180,E1 -16614.629,E2 -16614.629} C_VEL
LIN {X 0,Y 291.415,Z 76.335,A -85,B 0,C 180,E1 -16617.027,E2 -16617.027} C_VEL
LIN {X 0,Y 293.998,Z 88.511,A -85,B 0,C 180,E1 -16620.656,E2 -16620.656} C_VEL
LIN {X 0,Y 295.32,Z 95.896,A -85,B 0,C 180,E1 -16622.766,E2 -16622.766} C_VEL
LIN {X 0,Y 294.691,Z 102.77,A -85,B 0,C 180,E1 -16624.578,E2 -16624.578} C_VEL
LIN {X 0,Y 294.606,Z 103.493,A -85,B 0,C 180,E1 -16624.767,E2 -16624.767} C_VEL
LIN {X 0,Y 299.795,Z 146.157,A -85,B 0,C 180,E1 -16626.222,E2 -16626.222} C_VEL
LIN {X 0,Y 300.277,Z 151.887,A -85,B 0,C 180,E1 -16626.397,E2 -16626.397} C_VEL
LIN {X 0,Y 298.948,Z 212.642,A -85,B 0,C 180,E1 -16627.867,E2 -16627.867} C_VEL
LIN {X 0,Y 298.218,Z 225.762,A -85,B 0,C 180,E1 -16628.439,E2 -16628.439} C_VEL
LIN {X 0,Y 297.22,Z 237.983,A -85,B 0,C 180,E1 -16629.225,E2 -16629.225} C_VEL
LIN {X 0,Y 296.045,Z 249.496,A -85,B 0,C 180,E1 -16630.227,E2 -16630.227} C_VEL
LIN {X 0,Y 294.528,Z 261.296,A -85,B 0,C 180,E1 -16631.568,E2 -16631.568} C_VEL
LIN {X 0,Y 293.358,Z 271.941,A -85,B 0,C 180,E1 -16633.113,E2 -16633.113} C_VEL
LIN {X 0,Y 292.447,Z 279.164,A -85,B 0,C 180,E1 -16634.385,E2 -16634.385} C_VEL
LIN {X 0,Y 291.353,Z 288.611,A -85,B 0,C 180,E1 -16636.397,E2 -16636.397} C_VEL
LIN {X 0,Y 290.401,Z 296.384,A -85,B 0,C 180,E1 -16638.483,E2 -16638.483} C_VEL
LIN {X 0,Y 289.994,Z 301.712,A -85,B 0,C 180,E1 -16640.232,E2 -16640.232} C_VEL
LIN {X 0,Y 289.689,Z 306.852,A -85,B 0,C 180,E1 -16642.332,E2 -16642.332} C_VEL
LIN {X 0,Y 289.542,Z 311.507,A -85,B 0,C 180,E1 -16644.873,E2 -16644.873} C_VEL
LIN {X 0,Y 289.613,Z 314.461,A -85,B 0,C 180,E1 -16647.218,E2 -16647.218} C_VEL
LIN {X 0,Y 289.678,Z 315.652,A -85,B 0,C 180,E1 -16648.609,E2 -16648.609} C_VEL
LIN {X 0,Y 289.767,Z 316.392,A -85,B 0,C 180,E1 -16649.999,E2 -16649.999} C_VEL
LIN {X 0,Y 289.544,Z 316.654,A -85,B 0,C 180,E1 -16652.782,E2 -16652.782} C_VEL
LIN {X 0,Y 289.509,Z 316.206,A -85,B 0,C 180,E1 -16654.176,E2 -16654.176} C_VEL
LIN {X 0,Y 289.48,Z 315.332,A -85,B 0,C 180,E1 -16655.572,E2 -16655.572} C_VEL
LIN {X 0,Y 289.772,Z 312.371,A -85,B 0,C 180,E1 -16658.367,E2 -16658.367} C_VEL
LIN {X 0,Y 290.302,Z 309.032,A -85,B 0,C 180,E1 -16660.461,E2 -16660.461} C_VEL
LIN {X 0,Y 291.115,Z 304.647,A -85,B 0,C 180,E1 -16662.548,E2 -16662.548} C_VEL
LIN {X 0,Y 292.805,Z 298.079,A -85,B 0,C 180,E1 -16664.952,E2 -16664.952} C_VEL
LIN {X 0,Y 294.351,Z 291.194,A -85,B 0,C 180,E1 -16666.931,E2 -16666.931} C_VEL
LIN {X 0,Y 296.028,Z 283.668,A -85,B 0,C 180,E1 -16668.693,E2 -16668.693} C_VEL
LIN {X 0,Y 298.079,Z 274.925,A -85,B 0,C 180,E1 -16670.35,E2 -16670.35} C_VEL
LIN {X 0,Y 300.364,Z 264.202,A -85,B 0,C 180,E1 -16671.985,E2 -16671.985} C_VEL
LIN {X 0,Y 302.469,Z 253.528,A -85,B 0,C 180,E1 -16673.265,E2 -16673.265} C_VEL
LIN {X 0,Y 304.52,Z 241.587,A -85,B 0,C 180,E1 -16674.364,E2 -16674.364} C_VEL
LIN {X 0,Y 306.207,Z 229.196,A -85,B 0,C 180,E1 -16675.216,E2 -16675.216} C_VEL
LIN {X 0,Y 307.533,Z 215.935,A -85,B 0,C 180,E1 -16675.844,E2 -16675.844} C_VEL
LIN {X 0,Y 308.293,Z 199.707,A -85,B 0,C 180,E1 -16676.296,E2 -16676.296} C_VEL
LIN {X 0,Y 309.639,Z 153.176,A -85,B 0,C 180,E1 -16677.399,E2 -16677.399} C_VEL
LIN {X 0,Y 306.449,Z 132.847,A -85,B 0,C 180,E1 -16678.328,E2 -16678.328} C_VEL
LIN {X 0,Y 302.217,Z 112.29,A -85,B 0,C 180,E1 -16679.427,E2 -16679.427} C_VEL
LIN {X 0,Y 299.224,Z 105.508,A -85,B 0,C 180,E1 -16680.009,E2 -16680.009} C_VEL
LIN {X 0,Y 297.776,Z 101.976,A -85,B 0,C 180,E1 -16680.335,E2 -16680.335} C_VEL
LIN {X 0,Y 295.243,Z 90.716,A -85,B 0,C 180,E1 -16684.121,E2 -16684.121} C_VEL
LIN {X 0,Y 292.743,Z 81.145,A -85,B 0,C 180,E1 -16687.604,E2 -16687.604} C_VEL
LIN {X 0,Y 291.369,Z 76.192,A -85,B 0,C 180,E1 -16689.6,E2 -16689.6} C_VEL
LIN {X 0,Y 291.307,Z 76.198,A -85,B 0,C 180,E1 -16693.633,E2 -16693.633} C_VEL
LIN {X 0,Y 291.349,Z 76.191,A -85,B 0,C 180,E1 -16697.513,E2 -16697.513} C_VEL
LIN {X 0,Y 291.373,Z 76.191,A -85,B 0,C 180,E1 -16701.162,E2 -16701.162} C_VEL
LIN {X 0,Y 291.383,Z 76.188,A -85,B 0,C 180,E1 -16704.629,E2 -16704.629} C_VEL
LIN {X 0,Y 291.37,Z 76.19,A -85,B 0,C 180,E1 -16707.951,E2 -16707.951} C_VEL
LIN {X 0,Y 291.38,Z 76.191,A -85,B 0,C 180,E1 -16711.158,E2 -16711.158} C_VEL
LIN {X 0,Y 291.414,Z 76.179,A -85,B 0,C 180,E1 -16714.272,E2 -16714.272} C_VEL
LIN {X 0,Y 291.38,Z 76.177,A -85,B 0,C 180,E1 -16717.3,E2 -16717.3} C_VEL
LIN {X 0,Y 291.46,Z 76.18,A -85,B 0,C 180,E1 -16720.271,E2 -16720.271} C_VEL
LIN {X 0,Y 291.553,Z 76.169,A -85,B 0,C 180,E1 -16724.624,E2 -16724.624} C_VEL
LIN {X 0,Y 291.534,Z 76.169,A -85,B 0,C 180,E1 -16728.881,E2 -16728.881} C_VEL
LIN {X 0,Y 291.703,Z 76.139,A -85,B 0,C 180,E1 -16731.689,E2 -16731.689} C_VEL
LIN {X 0,Y 291.625,Z 76.159,A -85,B 0,C 180,E1 -16734.469,E2 -16734.469} C_VEL
LIN {X 0,Y 291.887,Z 76.118,A -85,B 0,C 180,E1 -16738.621,E2 -16738.621} C_VEL
LIN {X 0,Y 291.886,Z 76.122,A -85,B 0,C 180,E1 -16741.38,E2 -16741.38} C_VEL
LIN {X 0,Y 291.72,Z 76.141,A -85,B 0,C 180,E1 -16746.919,E2 -16746.919} C_VEL
LIN {X 0,Y 291.566,Z 76.164,A -85,B 0,C 180,E1 -16749.714,E2 -16749.714} C_VEL
LIN {X 0,Y 291.513,Z 76.167,A -85,B 0,C 180,E1 -16753.951,E2 -16753.951} C_VEL
LIN {X 0,Y 291.439,Z 76.174,A -85,B 0,C 180,E1 -16758.27,E2 -16758.27} C_VEL
LIN {X 0,Y 291.357,Z 76.183,A -85,B 0,C 180,E1 -16761.213,E2 -16761.213} C_VEL
LIN {X 0,Y 291.365,Z 76.192,A -85,B 0,C 180,E1 -16764.209,E2 -16764.209} C_VEL
LIN {X 0,Y 291.36,Z 76.193,A -85,B 0,C 180,E1 -16767.278,E2 -16767.278} C_VEL
LIN {X 0,Y 291.321,Z 76.196,A -85,B 0,C 180,E1 -16770.439,E2 -16770.439} C_VEL
LIN {X 0,Y 291.342,Z 76.194,A -85,B 0,C 180,E1 -16773.699,E2 -16773.699} C_VEL
LIN {X 0,Y 291.368,Z 76.191,A -85,B 0,C 180,E1 -16777.253,E2 -16777.253} C_VEL
LIN {X 0,Y 291.327,Z 76.186,A -85,B 0,C 180,E1 -16780.644,E2 -16780.644} C_VEL
LIN {X 0,Y 291.338,Z 76.31,A -85,B 0,C 180,E1 -16784.667,E2 -16784.667} C_VEL
LIN {X 0,Y 291.456,Z 76.956,A -85,B 0,C 180,E1 -16784.851,E2 -16784.851} C_VEL
LIN {X 0,Y 292.821,Z 79.748,A -85,B 0,C 180,E1 -16785.134,E2 -16785.134} C_VEL
LIN {X 0,Y 293.832,Z 81.154,A -85,B 0,C 180,E1 -16785.321,E2 -16785.321} C_VEL
LIN {X 0,Y 299.897,Z 91.874,A -85,B 0,C 180,E1 -16786.471,E2 -16786.471} C_VEL
LIN {X 0,Y 308.275,Z 108.889,A -85,B 0,C 180,E1 -16788.017,E2 -16788.017} C_VEL
LIN {X 0,Y 311.029,Z 115.204,A -85,B 0,C 180,E1 -16788.519,E2 -16788.519} C_VEL
LIN {X 0,Y 308.782,Z 181.397,A -85,B 0,C 180,E1 -16790.075,E2 -16790.075} C_VEL
LIN {X 0,Y 307.882,Z 194.386,A -85,B 0,C 180,E1 -16790.596,E2 -16790.596} C_VEL
LIN {X 0,Y 306.813,Z 207.088,A -85,B 0,C 180,E1 -16791.399,E2 -16791.399} C_VEL
LIN {X 0,Y 305.229,Z 219.008,A -85,B 0,C 180,E1 -16792.399,E2 -16792.399} C_VEL
LIN {X 0,Y 303.472,Z 229.921,A -85,B 0,C 180,E1 -16793.599,E2 -16793.599} C_VEL
LIN {X 0,Y 301.362,Z 241.027,A -85,B 0,C 180,E1 -16795.156,E2 -16795.156} C_VEL
LIN {X 0,Y 299.172,Z 250.913,A -85,B 0,C 180,E1 -16796.896,E2 -16796.896} C_VEL
LIN {X 0,Y 297.32,Z 258.901,A -85,B 0,C 180,E1 -16798.666,E2 -16798.666} C_VEL
LIN {X 0,Y 295.324,Z 266.625,A -85,B 0,C 180,E1 -16800.801,E2 -16800.801} C_VEL
LIN {X 0,Y 293.668,Z 272.751,A -85,B 0,C 180,E1 -16802.955,E2 -16802.955} C_VEL
LIN {X 0,Y 292.351,Z 277.516,A -85,B 0,C 180,E1 -16805.122,E2 -16805.122} C_VEL
LIN {X 0,Y 291.335,Z 281.08,A -85,B 0,C 180,E1 -16807.296,E2 -16807.296} C_VEL
LIN {X 0,Y 290.795,Z 282.826,A -85,B 0,C 180,E1 -16808.745,E2 -16808.745} C_VEL
LIN {X 0,Y 290.18,Z 284.586,A -85,B 0,C 180,E1 -16810.834,E2 -16810.834} C_VEL
LIN {X 0,Y 289.719,Z 285.467,A -85,B 0,C 180,E1 -16813.077,E2 -16813.077} C_VEL
LIN {X 0,Y 289.58,Z 285.481,A -85,B 0,C 180,E1 -16814.517,E2 -16814.517} C_VEL
LIN {X 0,Y 289.539,Z 285.025,A -85,B 0,C 180,E1 -16816.152,E2 -16816.152} C_VEL
LIN {X 0,Y 289.581,Z 283.075,A -85,B 0,C 180,E1 -16818.805,E2 -16818.805} C_VEL
LIN {X 0,Y 289.849,Z 280.441,A -85,B 0,C 180,E1 -16820.933,E2 -16820.933} C_VEL
LIN {X 0,Y 290.261,Z 276.704,A -85,B 0,C 180,E1 -16823.087,E2 -16823.087} C_VEL
LIN {X 0,Y 290.743,Z 272.024,A -85,B 0,C 180,E1 -16825.147,E2 -16825.147} C_VEL
LIN {X 0,Y 291.433,Z 266.007,A -85,B 0,C 180,E1 -16827.236,E2 -16827.236} C_VEL
LIN {X 0,Y 292.458,Z 258.506,A -85,B 0,C 180,E1 -16829.312,E2 -16829.312} C_VEL
LIN {X 0,Y 293.459,Z 250.863,A -85,B 0,C 180,E1 -16831.03,E2 -16831.03} C_VEL
LIN {X 0,Y 294.697,Z 241.568,A -85,B 0,C 180,E1 -16832.734,E2 -16832.734} C_VEL
LIN {X 0,Y 295.904,Z 231.33,A -85,B 0,C 180,E1 -16834.244,E2 -16834.244} C_VEL
LIN {X 0,Y 297.096,Z 219.777,A -85,B 0,C 180,E1 -16835.6,E2 -16835.6} C_VEL
LIN {X 0,Y 298.023,Z 207.833,A -85,B 0,C 180,E1 -16836.687,E2 -16836.687} C_VEL
LIN {X 0,Y 298.902,Z 194.511,A -85,B 0,C 180,E1 -16837.558,E2 -16837.558} C_VEL
LIN {X 0,Y 299.43,Z 181.672,A -85,B 0,C 180,E1 -16838.122,E2 -16838.122} C_VEL
LIN {X 0,Y 301.28,Z 103.652,A -85,B 0,C 180,E1 -16839.986,E2 -16839.986} C_VEL
LIN {X 0,Y 296.547,Z 88.991,A -85,B 0,C 180,E1 -16840.69,E2 -16840.69} C_VEL
LIN {X 0,Y 291.672,Z 76.916,A -85,B 0,C 180,E1 -16841.364,E2 -16841.364} C_VEL
LIN {X 0,Y 291.537,Z 76.171,A -85,B 0,C 180,E1 -16841.436,E2 -16841.436} C_VEL
LIN {X 0,Y 291.56,Z 76.168,A -85,B 0,C 180,E1 -16845.377,E2 -16845.377} C_VEL
LIN {X 0,Y 291.455,Z 76.179,A -85,B 0,C 180,E1 -16849.875,E2 -16849.875} C_VEL
LIN {X 0,Y 291.388,Z 76.191,A -85,B 0,C 180,E1 -16854.207,E2 -16854.207} C_VEL
LIN {X 0,Y 291.424,Z 76.179,A -85,B 0,C 180,E1 -16857.272,E2 -16857.272} C_VEL
LIN {X 0,Y 291.339,Z 76.193,A -85,B 0,C 180,E1 -16860.437,E2 -16860.437} C_VEL
LIN {X 0,Y 291.349,Z 76.189,A -85,B 0,C 180,E1 -16863.698,E2 -16863.698} C_VEL
LIN {X 0,Y 291.399,Z 76.186,A -85,B 0,C 180,E1 -16867.259,E2 -16867.259} C_VEL
LIN {X 0,Y 291.355,Z 76.189,A -85,B 0,C 180,E1 -16870.639,E2 -16870.639} C_VEL
LIN {X 0,Y 291.326,Z 76.192,A -85,B 0,C 180,E1 -16874.396,E2 -16874.396} C_VEL
LIN {X 0,Y 291.331,Z 76.193,A -85,B 0,C 180,E1 -16878.404,E2 -16878.404} C_VEL
LIN {X 0,Y 291.351,Z 76.189,A -85,B 0,C 180,E1 -16881.157,E2 -16881.157} C_VEL
LIN {X 0,Y 291.364,Z 76.176,A -85,B 0,C 180,E1 -16884.626,E2 -16884.626} C_VEL
LIN {X 0,Y 291.374,Z 76.183,A -85,B 0,C 180,E1 -16887.95,E2 -16887.95} C_VEL
LIN {X 0,Y 291.373,Z 76.188,A -85,B 0,C 180,E1 -16891.903,E2 -16891.903} C_VEL
LIN {X 0,Y 290.724,Z 76.271,A -85,B 0,C 180,E1 -16893.058,E2 -16893.058} C_VEL
LIN {X 0,Y 287.858,Z 76.623,A -85,B 0,C 180,E1 -16894.937,E2 -16894.937} C_VEL
LIN {X 0,Y 285.425,Z 76.927,A -85,B 0,C 180,E1 -16896.463,E2 -16896.463} C_VEL
LIN {X 0,Y 284.399,Z 77.055,A -85,B 0,C 180,E1 -16897.646,E2 -16897.646} C_VEL
LIN {X 0,Y 284.325,Z 77.065,A -85,B 0,C 180,E1 -16898.047,E2 -16898.047} C_VEL
LIN {X 0,Y 284.406,Z 77.055,A -85,B 0,C 180,E1 -16901.261,E2 -16901.261} C_VEL
LIN {X 0,Y 284.495,Z 77.045,A -85,B 0,C 180,E1 -16904.459,E2 -16904.459} C_VEL
LIN {X 0,Y 284.49,Z 77.046,A -85,B 0,C 180,E1 -16908.601,E2 -16908.601} C_VEL
LIN {X 0,Y 284.642,Z 77.024,A -85,B 0,C 180,E1 -16911.48,E2 -16911.48} C_VEL
LIN {X 0,Y 284.599,Z 77.033,A -85,B 0,C 180,E1 -16914.331,E2 -16914.331} C_VEL
LIN {X 0,Y 284.857,Z 76.997,A -85,B 0,C 180,E1 -16918.586,E2 -16918.586} C_VEL
LIN {X 0,Y 284.857,Z 76.998,A -85,B 0,C 180,E1 -16921.413,E2 -16921.413} C_VEL
LIN {X 0,Y 284.676,Z 77.022,A -85,B 0,C 180,E1 -16927.09,E2 -16927.09} C_VEL
LIN {X 0,Y 284.516,Z 77.043,A -85,B 0,C 180,E1 -16929.957,E2 -16929.957} C_VEL
LIN {X 0,Y 284.484,Z 77.044,A -85,B 0,C 180,E1 -16934.302,E2 -16934.302} C_VEL
LIN {X 0,Y 284.427,Z 77.056,A -85,B 0,C 180,E1 -16937.248,E2 -16937.248} C_VEL
LIN {X 0,Y 284.379,Z 77.059,A -85,B 0,C 180,E1 -16940.242,E2 -16940.242} C_VEL
LIN {X 0,Y 284.338,Z 77.068,A -85,B 0,C 180,E1 -16944.846,E2 -16944.846} C_VEL
LIN {X 0,Y 284.332,Z 77.065,A -85,B 0,C 180,E1 -16948.01,E2 -16948.01} C_VEL
LIN {X 0,Y 284.297,Z 77.068,A -85,B 0,C 180,E1 -16951.274,E2 -16951.274} C_VEL
LIN {X 0,Y 284.343,Z 77.064,A -85,B 0,C 180,E1 -16955.348,E2 -16955.348} C_VEL
LIN {X 0,Y 284.314,Z 77.07,A -85,B 0,C 180,E1 -16958.169,E2 -16958.169} C_VEL
LIN {X 0,Y 284.271,Z 77.076,A -85,B 0,C 180,E1 -16962.124,E2 -16962.124} C_VEL
LIN {X 0,Y 284.257,Z 77.077,A -85,B 0,C 180,E1 -16966.189,E2 -16966.189} C_VEL
LIN {X 0,Y 284.309,Z 77.072,A -85,B 0,C 180,E1 -16970.023,E2 -16970.023} C_VEL
LIN {X 0,Y 284.352,Z 77.067,A -85,B 0,C 180,E1 -16973.616,E2 -16973.616} C_VEL
LIN {X 0,Y 284.37,Z 77.222,A -85,B 0,C 180,E1 -16976.641,E2 -16976.641} C_VEL
LIN {X 0,Y 287.163,Z 90.477,A -85,B 0,C 180,E1 -16980.693,E2 -16980.693} C_VEL
LIN {X 0,Y 288.376,Z 97.732,A -85,B 0,C 180,E1 -16982.809,E2 -16982.809} C_VEL
LIN {X 0,Y 287.771,Z 103.158,A -85,B 0,C 180,E1 -16984.27,E2 -16984.27} C_VEL
LIN {X 0,Y 293.151,Z 147.289,A -85,B 0,C 180,E1 -16985.808,E2 -16985.808} C_VEL
LIN {X 0,Y 293.537,Z 153.035,A -85,B 0,C 180,E1 -16985.982,E2 -16985.982} C_VEL
LIN {X 0,Y 292.187,Z 212.577,A -85,B 0,C 180,E1 -16987.458,E2 -16987.458} C_VEL
LIN {X 0,Y 291.342,Z 226.497,A -85,B 0,C 180,E1 -16988.09,E2 -16988.09} C_VEL
LIN {X 0,Y 290.248,Z 239.485,A -85,B 0,C 180,E1 -16988.981,E2 -16988.981} C_VEL
LIN {X 0,Y 288.883,Z 251.298,A -85,B 0,C 180,E1 -16990.086,E2 -16990.086} C_VEL
LIN {X 0,Y 287.442,Z 262.705,A -85,B 0,C 180,E1 -16991.466,E2 -16991.466} C_VEL
LIN {X 0,Y 286.381,Z 271.957,A -85,B 0,C 180,E1 -16992.873,E2 -16992.873} C_VEL
LIN {X 0,Y 285.405,Z 279.664,A -85,B 0,C 180,E1 -16994.283,E2 -16994.283} C_VEL
LIN {X 0,Y 284.382,Z 287.749,A -85,B 0,C 180,E1 -16996.057,E2 -16996.057} C_VEL
LIN {X 0,Y 283.414,Z 295.643,A -85,B 0,C 180,E1 -16998.195,E2 -16998.195} C_VEL
LIN {X 0,Y 282.819,Z 302.879,A -85,B 0,C 180,E1 -17000.704,E2 -17000.704} C_VEL
LIN {X 0,Y 282.561,Z 307.686,A -85,B 0,C 180,E1 -17002.856,E2 -17002.856} C_VEL
LIN {X 0,Y 282.483,Z 310.39,A -85,B 0,C 180,E1 -17004.37,E2 -17004.37} C_VEL
LIN {X 0,Y 282.513,Z 312.33,A -85,B 0,C 180,E1 -17005.72,E2 -17005.72} C_VEL
LIN {X 0,Y 282.535,Z 313.962,A -85,B 0,C 180,E1 -17007.148,E2 -17007.148} C_VEL
LIN {X 0,Y 282.587,Z 315.183,A -85,B 0,C 180,E1 -17008.574,E2 -17008.574} C_VEL
LIN {X 0,Y 282.676,Z 315.969,A -85,B 0,C 180,E1 -17009.999,E2 -17009.999} C_VEL
LIN {X 0,Y 282.468,Z 316.281,A -85,B 0,C 180,E1 -17012.852,E2 -17012.852} C_VEL
LIN {X 0,Y 282.39,Z 315.213,A -85,B 0,C 180,E1 -17015.436,E2 -17015.436} C_VEL
LIN {X 0,Y 282.492,Z 313.775,A -85,B 0,C 180,E1 -17017.145,E2 -17017.145} C_VEL
LIN {X 0,Y 283.07,Z 310.061,A -85,B 0,C 180,E1 -17020.008,E2 -17020.008} C_VEL
LIN {X 0,Y 283.814,Z 306.092,A -85,B 0,C 180,E1 -17022.15,E2 -17022.15} C_VEL
LIN {X 0,Y 285.11,Z 301.023,A -85,B 0,C 180,E1 -17024.27,E2 -17024.27} C_VEL
LIN {X 0,Y 286.669,Z 294.693,A -85,B 0,C 180,E1 -17026.375,E2 -17026.375} C_VEL
LIN {X 0,Y 288.566,Z 286.813,A -85,B 0,C 180,E1 -17028.458,E2 -17028.458} C_VEL
LIN {X 0,Y 290.565,Z 278.819,A -85,B 0,C 180,E1 -17030.161,E2 -17030.161} C_VEL
LIN {X 0,Y 292.853,Z 269.099,A -85,B 0,C 180,E1 -17031.837,E2 -17031.837} C_VEL
LIN {X 0,Y 294.988,Z 259.609,A -85,B 0,C 180,E1 -17033.147,E2 -17033.147} C_VEL
LIN {X 0,Y 296.907,Z 249.462,A -85,B 0,C 180,E1 -17034.285,E2 -17034.285} C_VEL
LIN {X 0,Y 298.898,Z 237.514,A -85,B 0,C 180,E1 -17035.317,E2 -17035.317} C_VEL
LIN {X 0,Y 300.625,Z 224.272,A -85,B 0,C 180,E1 -17036.137,E2 -17036.137} C_VEL
LIN {X 0,Y 301.771,Z 210.862,A -85,B 0,C 180,E1 -17036.692,E2 -17036.692} C_VEL
LIN {X 0,Y 303.599,Z 154.201,A -85,B 0,C 180,E1 -17038.078,E2 -17038.078} C_VEL
LIN {X 0,Y 300.628,Z 134.887,A -85,B 0,C 180,E1 -17038.987,E2 -17038.987} C_VEL
LIN {X 0,Y 296.513,Z 114.666,A -85,B 0,C 180,E1 -17040.103,E2 -17040.103} C_VEL
LIN {X 0,Y 291.551,Z 104.171,A -85,B 0,C 180,E1 -17041.096,E2 -17041.096} C_VEL
LIN {X 0,Y 290.466,Z 101.543,A -85,B 0,C 180,E1 -17041.348,E2 -17041.348} C_VEL
LIN {X 0,Y 288.418,Z 92.453,A -85,B 0,C 180,E1 -17044.508,E2 -17044.508} C_VEL
LIN {X 0,Y 286.094,Z 83.434,A -85,B 0,C 180,E1 -17047.888,E2 -17047.888} C_VEL
LIN {X 0,Y 284.304,Z 77.07,A -85,B 0,C 180,E1 -17050.457,E2 -17050.457} C_VEL
LIN {X 0,Y 284.243,Z 77.068,A -85,B 0,C 180,E1 -17054.19,E2 -17054.19} C_VEL
LIN {X 0,Y 284.3,Z 77.072,A -85,B 0,C 180,E1 -17058.13,E2 -17058.13} C_VEL
LIN {X 0,Y 284.327,Z 77.062,A -85,B 0,C 180,E1 -17061.834,E2 -17061.834} C_VEL
LIN {X 0,Y 284.321,Z 77.062,A -85,B 0,C 180,E1 -17065.353,E2 -17065.353} C_VEL
LIN {X 0,Y 284.294,Z 77.066,A -85,B 0,C 180,E1 -17068.726,E2 -17068.726} C_VEL
LIN {X 0,Y 284.395,Z 77.051,A -85,B 0,C 180,E1 -17072.826,E2 -17072.826} C_VEL
LIN {X 0,Y 284.364,Z 77.054,A -85,B 0,C 180,E1 -17076.707,E2 -17076.707} C_VEL
LIN {X 0,Y 284.403,Z 77.051,A -85,B 0,C 180,E1 -17081.262,E2 -17081.262} C_VEL
LIN {X 0,Y 284.49,Z 77.049,A -85,B 0,C 180,E1 -17084.459,E2 -17084.459} C_VEL
LIN {X 0,Y 284.486,Z 77.042,A -85,B 0,C 180,E1 -17088.602,E2 -17088.602} C_VEL
LIN {X 0,Y 284.654,Z 77.018,A -85,B 0,C 180,E1 -17091.481,E2 -17091.481} C_VEL
LIN {X 0,Y 284.596,Z 77.034,A -85,B 0,C 180,E1 -17094.331,E2 -17094.331} C_VEL
LIN {X 0,Y 284.853,Z 76.993,A -85,B 0,C 180,E1 -17098.587,E2 -17098.587} C_VEL
LIN {X 0,Y 284.852,Z 76.998,A -85,B 0,C 180,E1 -17101.414,E2 -17101.414} C_VEL
LIN {X 0,Y 284.671,Z 77.016,A -85,B 0,C 180,E1 -17107.091,E2 -17107.091} C_VEL
LIN {X 0,Y 284.512,Z 77.045,A -85,B 0,C 180,E1 -17109.958,E2 -17109.958} C_VEL
LIN {X 0,Y 284.461,Z 77.048,A -85,B 0,C 180,E1 -17114.304,E2 -17114.304} C_VEL
LIN {X 0,Y 284.373,Z 77.057,A -85,B 0,C 180,E1 -17118.741,E2 -17118.741} C_VEL
LIN {X 0,Y 284.313,Z 77.059,A -85,B 0,C 180,E1 -17121.765,E2 -17121.765} C_VEL
LIN {X 0,Y 284.314,Z 77.064,A -85,B 0,C 180,E1 -17124.849,E2 -17124.849} C_VEL
LIN {X 0,Y 284.29,Z 77.074,A -85,B 0,C 180,E1 -17128.016,E2 -17128.016} C_VEL
LIN {X 0,Y 284.285,Z 77.073,A -85,B 0,C 180,E1 -17131.276,E2 -17131.276} C_VEL
LIN {X 0,Y 284.339,Z 77.061,A -85,B 0,C 180,E1 -17135.349,E2 -17135.349} C_VEL
LIN {X 0,Y 284.305,Z 77.071,A -85,B 0,C 180,E1 -17138.171,E2 -17138.171} C_VEL
LIN {X 0,Y 284.264,Z 77.069,A -85,B 0,C 180,E1 -17142.124,E2 -17142.124} C_VEL
LIN {X 0,Y 284.268,Z 77.146,A -85,B 0,C 180,E1 -17143.752,E2 -17143.752} C_VEL
LIN {X 0,Y 285.297,Z 79.988,A -85,B 0,C 180,E1 -17144.02,E2 -17144.02} C_VEL
LIN {X 0,Y 287.09,Z 82.547,A -85,B 0,C 180,E1 -17144.374,E2 -17144.374} C_VEL
LIN {X 0,Y 292.719,Z 91.96,A -85,B 0,C 180,E1 -17145.489,E2 -17145.489} C_VEL
LIN {X 0,Y 301.253,Z 108.826,A -85,B 0,C 180,E1 -17147.135,E2 -17147.135} C_VEL
LIN {X 0,Y 304.975,Z 117.171,A -85,B 0,C 180,E1 -17147.843,E2 -17147.843} C_VEL
LIN {X 0,Y 302.707,Z 181.93,A -85,B 0,C 180,E1 -17149.397,E2 -17149.397} C_VEL
LIN {X 0,Y 301.766,Z 195.075,A -85,B 0,C 180,E1 -17149.94,E2 -17149.94} C_VEL
LIN {X 0,Y 300.683,Z 207.307,A -85,B 0,C 180,E1 -17150.727,E2 -17150.727} C_VEL
LIN {X 0,Y 299.086,Z 218.836,A -85,B 0,C 180,E1 -17151.702,E2 -17151.702} C_VEL
LIN {X 0,Y 297.271,Z 229.905,A -85,B 0,C 180,E1 -17152.925,E2 -17152.925} C_VEL
LIN {X 0,Y 295.122,Z 240.643,A -85,B 0,C 180,E1 -17154.437,E2 -17154.437} C_VEL
LIN {X 0,Y 292.952,Z 250.105,A -85,B 0,C 180,E1 -17156.099,E2 -17156.099} C_VEL
LIN {X 0,Y 290.973,Z 258.343,A -85,B 0,C 180,E1 -17157.902,E2 -17157.902} C_VEL
LIN {X 0,Y 288.872,Z 266.263,A -85,B 0,C 180,E1 -17160.084,E2 -17160.084} C_VEL
LIN {X 0,Y 287.033,Z 272.532,A -85,B 0,C 180,E1 -17162.277,E2 -17162.277} C_VEL
LIN {X 0,Y 285.609,Z 277.43,A -85,B 0,C 180,E1 -17164.493,E2 -17164.493} C_VEL
LIN {X 0,Y 284.514,Z 281.117,A -85,B 0,C 180,E1 -17166.72,E2 -17166.72} C_VEL
LIN {X 0,Y 283.899,Z 282.975,A -85,B 0,C 180,E1 -17168.203,E2 -17168.203} C_VEL
LIN {X 0,Y 283.144,Z 284.981,A -85,B 0,C 180,E1 -17170.6,E2 -17170.6} C_VEL
LIN {X 0,Y 282.693,Z 285.822,A -85,B 0,C 180,E1 -17172.643,E2 -17172.643} C_VEL
LIN {X 0,Y 282.517,Z 285.902,A -85,B 0,C 180,E1 -17174.12,E2 -17174.12} C_VEL
LIN {X 0,Y 282.452,Z 285.417,A -85,B 0,C 180,E1 -17176.028,E2 -17176.028} C_VEL
LIN {X 0,Y 282.483,Z 283.71,A -85,B 0,C 180,E1 -17178.52,E2 -17178.52} C_VEL
LIN {X 0,Y 282.735,Z 281.184,A -85,B 0,C 180,E1 -17180.702,E2 -17180.702} C_VEL
LIN {X 0,Y 283.169,Z 277.175,A -85,B 0,C 180,E1 -17183.108,E2 -17183.108} C_VEL
LIN {X 0,Y 283.615,Z 273.014,A -85,B 0,C 180,E1 -17185.025,E2 -17185.025} C_VEL
LIN {X 0,Y 284.461,Z 266.011,A -85,B 0,C 180,E1 -17187.522,E2 -17187.522} C_VEL
LIN {X 0,Y 285.518,Z 258.432,A -85,B 0,C 180,E1 -17189.648,E2 -17189.648} C_VEL
LIN {X 0,Y 286.587,Z 250.686,A -85,B 0,C 180,E1 -17191.406,E2 -17191.406} C_VEL
LIN {X 0,Y 288.007,Z 240.152,A -85,B 0,C 180,E1 -17193.323,E2 -17193.323} C_VEL
LIN {X 0,Y 289.299,Z 229.418,A -85,B 0,C 180,E1 -17194.881,E2 -17194.881} C_VEL
LIN {X 0,Y 290.371,Z 219.068,A -85,B 0,C 180,E1 -17196.079,E2 -17196.079} C_VEL
LIN {X 0,Y 291.34,Z 206.669,A -85,B 0,C 180,E1 -17197.189,E2 -17197.189} C_VEL
LIN {X 0,Y 292.208,Z 193.566,A -85,B 0,C 180,E1 -17198.037,E2 -17198.037} C_VEL
LIN {X 0,Y 292.737,Z 180.911,A -85,B 0,C 180,E1 -17198.574,E2 -17198.574} C_VEL
LIN {X 0,Y 294.496,Z 104.602,A -85,B 0,C 180,E1 -17200.437,E2 -17200.437} C_VEL
LIN {X 0,Y 289.25,Z 88.808,A -85,B 0,C 180,E1 -17201.235,E2 -17201.235} C_VEL
LIN {X 0,Y 284.514,Z 77.316,A -85,B 0,C 180,E1 -17201.907,E2 -17201.907} C_VEL
LIN {X 0,Y 284.497,Z 77.05,A -85,B 0,C 180,E1 -17201.941,E2 -17201.941} C_VEL
LIN {X 0,Y 284.492,Z 77.05,A -85,B 0,C 180,E1 -17205.768,E2 -17205.768} C_VEL
LIN {X 0,Y 284.382,Z 77.063,A -85,B 0,C 180,E1 -17210.242,E2 -17210.242} C_VEL
LIN {X 0,Y 284.343,Z 77.065,A -85,B 0,C 180,E1 -17214.847,E2 -17214.847} C_VEL
LIN {X 0,Y 284.333,Z 77.065,A -85,B 0,C 180,E1 -17218.011,E2 -17218.011} C_VEL
LIN {X 0,Y 284.299,Z 77.07,A -85,B 0,C 180,E1 -17221.274,E2 -17221.274} C_VEL
LIN {X 0,Y 284.366,Z 77.059,A -85,B 0,C 180,E1 -17225.354,E2 -17225.354} C_VEL
LIN {X 0,Y 284.328,Z 77.066,A -85,B 0,C 180,E1 -17228.167,E2 -17228.167} C_VEL
LIN {X 0,Y 284.3,Z 77.069,A -85,B 0,C 180,E1 -17232.13,E2 -17232.13} C_VEL
LIN {X 0,Y 284.272,Z 77.071,A -85,B 0,C 180,E1 -17236.192,E2 -17236.192} C_VEL
LIN {X 0,Y 284.31,Z 77.065,A -85,B 0,C 180,E1 -17240.024,E2 -17240.024} C_VEL
LIN {X 0,Y 284.334,Z 77.05,A -85,B 0,C 180,E1 -17243.614,E2 -17243.614} C_VEL
LIN {X 0,Y 284.311,Z 77.064,A -85,B 0,C 180,E1 -17247.19,E2 -17247.19} C_VEL
LIN {X 0,Y 284.359,Z 77.062,A -85,B 0,C 180,E1 -17250.375,E2 -17250.375} C_VEL
LIN {X 0,Y 284.378,Z 77.058,A -85,B 0,C 180,E1 -17253.586,E2 -17253.586} C_VEL
LIN {X 0,Y 284.37,Z 77.061,A -85,B 0,C 180,E1 -17256.707,E2 -17256.707} C_VEL
LIN {X 0,Y 284.325,Z 77.065,A -85,B 0,C 180,E1 -17258.047,E2 -17258.047} C_VEL
LIN {X 0,Y 283.708,Z 77.148,A -85,B 0,C 180,E1 -17259.23,E2 -17259.23} C_VEL
LIN {X 0,Y 280.952,Z 77.495,A -85,B 0,C 180,E1 -17261.159,E2 -17261.159} C_VEL
LIN {X 0,Y 278.581,Z 77.787,A -85,B 0,C 180,E1 -17262.725,E2 -17262.725} C_VEL
LIN {X 0,Y 277.54,Z 77.911,A -85,B 0,C 180,E1 -17263.937,E2 -17263.937} C_VEL
LIN {X 0,Y 277.443,Z 77.921,A -85,B 0,C 180,E1 -17264.347,E2 -17264.347} C_VEL
LIN {X 0,Y 277.437,Z 77.927,A -85,B 0,C 180,E1 -17268.307,E2 -17268.307} C_VEL
LIN {X 0,Y 277.601,Z 77.9,A -85,B 0,C 180,E1 -17271.262,E2 -17271.262} C_VEL
LIN {X 0,Y 277.57,Z 77.91,A -85,B 0,C 180,E1 -17274.187,E2 -17274.187} C_VEL
LIN {X 0,Y 277.823,Z 77.873,A -85,B 0,C 180,E1 -17278.55,E2 -17278.55} C_VEL
LIN {X 0,Y 277.823,Z 77.874,A -85,B 0,C 180,E1 -17281.449,E2 -17281.449} C_VEL
LIN {X 0,Y 277.63,Z 77.901,A -85,B 0,C 180,E1 -17287.271,E2 -17287.271} C_VEL
LIN {X 0,Y 277.46,Z 77.921,A -85,B 0,C 180,E1 -17290.213,E2 -17290.213} C_VEL
LIN {X 0,Y 277.437,Z 77.923,A -85,B 0,C 180,E1 -17294.674,E2 -17294.674} C_VEL
LIN {X 0,Y 277.347,Z 77.939,A -85,B 0,C 180,E1 -17299.233,E2 -17299.233} C_VEL
LIN {X 0,Y 277.293,Z 77.942,A -85,B 0,C 180,E1 -17304.157,E2 -17304.157} C_VEL
LIN {X 0,Y 277.326,Z 77.938,A -85,B 0,C 180,E1 -17307.504,E2 -17307.504} C_VEL
LIN {X 0,Y 277.274,Z 77.943,A -85,B 0,C 180,E1 -17310.481,E2 -17310.481} C_VEL
LIN {X 0,Y 277.249,Z 77.948,A -85,B 0,C 180,E1 -17313.895,E2 -17313.895} C_VEL
LIN {X 0,Y 277.269,Z 77.945,A -85,B 0,C 180,E1 -17317.469,E2 -17317.469} C_VEL
LIN {X 0,Y 277.211,Z 77.953,A -85,B 0,C 180,E1 -17321.236,E2 -17321.236} C_VEL
LIN {X 0,Y 277.202,Z 77.95,A -85,B 0,C 180,E1 -17325.226,E2 -17325.226} C_VEL
LIN {X 0,Y 277.224,Z 77.953,A -85,B 0,C 180,E1 -17329.512,E2 -17329.512} C_VEL
LIN {X 0,Y 277.283,Z 77.947,A -85,B 0,C 180,E1 -17332.533,E2 -17332.533} C_VEL
LIN {X 0,Y 277.308,Z 77.995,A -85,B 0,C 180,E1 -17336.206,E2 -17336.206} C_VEL
LIN {X 0,Y 279.99,Z 90.812,A -85,B 0,C 180,E1 -17340.237,E2 -17340.237} C_VEL
LIN {X 0,Y 281.354,Z 98.256,A -85,B 0,C 180,E1 -17342.476,E2 -17342.476} C_VEL
LIN {X 0,Y 280.974,Z 102.775,A -85,B 0,C 180,E1 -17343.733,E2 -17343.733} C_VEL
LIN {X 0,Y 286.136,Z 144.831,A -85,B 0,C 180,E1 -17345.256,E2 -17345.256} C_VEL
LIN {X 0,Y 286.854,Z 153.141,A -85,B 0,C 180,E1 -17345.526,E2 -17345.526} C_VEL
LIN {X 0,Y 285.429,Z 212.579,A -85,B 0,C 180,E1 -17347.038,E2 -17347.038} C_VEL
LIN {X 0,Y 284.562,Z 226.372,A -85,B 0,C 180,E1 -17347.683,E2 -17347.683} C_VEL
LIN {X 0,Y 283.464,Z 238.767,A -85,B 0,C 180,E1 -17348.549,E2 -17348.549} C_VEL
LIN {X 0,Y 281.983,Z 251.456,A -85,B 0,C 180,E1 -17349.768,E2 -17349.768} C_VEL
LIN {X 0,Y 280.503,Z 262.768,A -85,B 0,C 180,E1 -17351.18,E2 -17351.18} C_VEL
LIN {X 0,Y 279.211,Z 273.119,A -85,B 0,C 180,E1 -17352.828,E2 -17352.828} C_VEL
LIN {X 0,Y 278.129,Z 282.164,A -85,B 0,C 180,E1 -17354.613,E2 -17354.613} C_VEL
LIN {X 0,Y 277.103,Z 289.738,A -85,B 0,C 180,E1 -17356.431,E2 -17356.431} C_VEL
LIN {X 0,Y 276.148,Z 297.162,A -85,B 0,C 180,E1 -17358.624,E2 -17358.624} C_VEL
LIN {X 0,Y 275.759,Z 302.2,A -85,B 0,C 180,E1 -17360.464,E2 -17360.464} C_VEL
LIN {X 0,Y 275.488,Z 307.073,A -85,B 0,C 180,E1 -17362.671,E2 -17362.671} C_VEL
LIN {X 0,Y 275.392,Z 310.139,A -85,B 0,C 180,E1 -17364.432,E2 -17364.432} C_VEL
LIN {X 0,Y 275.458,Z 313.463,A -85,B 0,C 180,E1 -17367.075,E2 -17367.075} C_VEL
LIN {X 0,Y 275.499,Z 314.709,A -85,B 0,C 180,E1 -17368.538,E2 -17368.538} C_VEL
LIN {X 0,Y 275.586,Z 315.542,A -85,B 0,C 180,E1 -17369.999,E2 -17369.999} C_VEL
LIN {X 0,Y 275.391,Z 315.908,A -85,B 0,C 180,E1 -17372.925,E2 -17372.925} C_VEL
LIN {X 0,Y 275.296,Z 314.723,A -85,B 0,C 180,E1 -17375.86,E2 -17375.86} C_VEL
LIN {X 0,Y 275.422,Z 313.506,A -85,B 0,C 180,E1 -17377.33,E2 -17377.33} C_VEL
LIN {X 0,Y 275.853,Z 310.939,A -85,B 0,C 180,E1 -17379.532,E2 -17379.532} C_VEL
LIN {X 0,Y 276.507,Z 307.38,A -85,B 0,C 180,E1 -17381.732,E2 -17381.732} C_VEL
LIN {X 0,Y 277.73,Z 302.755,A -85,B 0,C 180,E1 -17383.91,E2 -17383.91} C_VEL
LIN {X 0,Y 279.278,Z 296.922,A -85,B 0,C 180,E1 -17386.07,E2 -17386.07} C_VEL
LIN {X 0,Y 280.963,Z 290.114,A -85,B 0,C 180,E1 -17388.097,E2 -17388.097} C_VEL
LIN {X 0,Y 283.009,Z 282.339,A -85,B 0,C 180,E1 -17389.965,E2 -17389.965} C_VEL
LIN {X 0,Y 285.315,Z 273.487,A -85,B 0,C 180,E1 -17391.683,E2 -17391.683} C_VEL
LIN {X 0,Y 287.872,Z 262.625,A -85,B 0,C 180,E1 -17393.373,E2 -17393.373} C_VEL
LIN {X 0,Y 290.175,Z 251.69,A -85,B 0,C 180,E1 -17394.695,E2 -17394.695} C_VEL
LIN {X 0,Y 292.371,Z 239.48,A -85,B 0,C 180,E1 -17395.828,E2 -17395.828} C_VEL
LIN {X 0,Y 294.193,Z 226.66,A -85,B 0,C 180,E1 -17396.705,E2 -17396.705} C_VEL
LIN {X 0,Y 295.522,Z 213.428,A -85,B 0,C 180,E1 -17397.307,E2 -17397.307} C_VEL
LIN {X 0,Y 296.344,Z 193.894,A -85,B 0,C 180,E1 -17397.841,E2 -17397.841} C_VEL
LIN {X 0,Y 297.565,Z 154.909,A -85,B 0,C 180,E1 -17398.803,E2 -17398.803} C_VEL
LIN {X 0,Y 294.732,Z 136.235,A -85,B 0,C 180,E1 -17399.711,E2 -17399.711} C_VEL
LIN {X 0,Y 291.02,Z 117.711,A -85,B 0,C 180,E1 -17400.763,E2 -17400.763} C_VEL
LIN {X 0,Y 285.02,Z 105.021,A -85,B 0,C 180,E1 -17402.022,E2 -17402.022} C_VEL
LIN {X 0,Y 283.185,Z 101,A -85,B 0,C 180,E1 -17402.456,E2 -17402.456} C_VEL
LIN {X 0,Y 280.96,Z 91.42,A -85,B 0,C 180,E1 -17405.955,E2 -17405.955} C_VEL
LIN {X 0,Y 278.63,Z 82.609,A -85,B 0,C 180,E1 -17409.454,E2 -17409.454} C_VEL
LIN {X 0,Y 277.232,Z 77.953,A -85,B 0,C 180,E1 -17411.473,E2 -17411.473} C_VEL
LIN {X 0,Y 277.204,Z 77.935,A -85,B 0,C 180,E1 -17415.225,E2 -17415.225} C_VEL
LIN {X 0,Y 277.26,Z 77.943,A -85,B 0,C 180,E1 -17419.502,E2 -17419.502} C_VEL
LIN {X 0,Y 277.283,Z 77.938,A -85,B 0,C 180,E1 -17422.533,E2 -17422.533} C_VEL
LIN {X 0,Y 277.252,Z 77.942,A -85,B 0,C 180,E1 -17426.105,E2 -17426.105} C_VEL
LIN {X 0,Y 277.259,Z 77.94,A -85,B 0,C 180,E1 -17429.538,E2 -17429.538} C_VEL
LIN {X 0,Y 277.356,Z 77.927,A -85,B 0,C 180,E1 -17432.864,E2 -17432.864} C_VEL
LIN {X 0,Y 277.327,Z 77.939,A -85,B 0,C 180,E1 -17436.08,E2 -17436.08} C_VEL
LIN {X 0,Y 277.344,Z 77.933,A -85,B 0,C 180,E1 -17440.766,E2 -17440.766} C_VEL
LIN {X 0,Y 277.432,Z 77.925,A -85,B 0,C 180,E1 -17445.326,E2 -17445.326} C_VEL
LIN {X 0,Y 277.504,Z 77.919,A -85,B 0,C 180,E1 -17449.789,E2 -17449.789} C_VEL
LIN {X 0,Y 277.647,Z 77.886,A -85,B 0,C 180,E1 -17452.729,E2 -17452.729} C_VEL
LIN {X 0,Y 277.819,Z 77.869,A -85,B 0,C 180,E1 -17458.551,E2 -17458.551} C_VEL
LIN {X 0,Y 277.818,Z 77.873,A -85,B 0,C 180,E1 -17461.45,E2 -17461.45} C_VEL
LIN {X 0,Y 277.625,Z 77.892,A -85,B 0,C 180,E1 -17467.272,E2 -17467.272} C_VEL
LIN {X 0,Y 277.455,Z 77.924,A -85,B 0,C 180,E1 -17470.214,E2 -17470.214} C_VEL
LIN {X 0,Y 277.408,Z 77.928,A -85,B 0,C 180,E1 -17474.676,E2 -17474.676} C_VEL
LIN {X 0,Y 277.323,Z 77.94,A -85,B 0,C 180,E1 -17479.236,E2 -17479.236} C_VEL
LIN {X 0,Y 277.286,Z 77.945,A -85,B 0,C 180,E1 -17483.925,E2 -17483.925} C_VEL
LIN {X 0,Y 277.279,Z 77.946,A -85,B 0,C 180,E1 -17487.488,E2 -17487.488} C_VEL
LIN {X 0,Y 277.246,Z 77.949,A -85,B 0,C 180,E1 -17490.473,E2 -17490.473} C_VEL
LIN {X 0,Y 277.245,Z 77.951,A -85,B 0,C 180,E1 -17493.897,E2 -17493.897} C_VEL
LIN {X 0,Y 277.262,Z 77.947,A -85,B 0,C 180,E1 -17497.471,E2 -17497.471} C_VEL
LIN {X 0,Y 277.231,Z 77.943,A -85,B 0,C 180,E1 -17501.979,E2 -17501.979} C_VEL
LIN {X 0,Y 277.239,Z 77.976,A -85,B 0,C 180,E1 -17502.665,E2 -17502.665} C_VEL
LIN {X 0,Y 278.285,Z 80.883,A -85,B 0,C 180,E1 -17502.934,E2 -17502.934} C_VEL
LIN {X 0,Y 280.014,Z 83.275,A -85,B 0,C 180,E1 -17503.293,E2 -17503.293} C_VEL
LIN {X 0,Y 287.019,Z 94.765,A -85,B 0,C 180,E1 -17504.744,E2 -17504.744} C_VEL
LIN {X 0,Y 294.475,Z 109.281,A -85,B 0,C 180,E1 -17506.248,E2 -17506.248} C_VEL
LIN {X 0,Y 298.95,Z 119.136,A -85,B 0,C 180,E1 -17507.132,E2 -17507.132} C_VEL
LIN {X 0,Y 296.692,Z 182.103,A -85,B 0,C 180,E1 -17508.675,E2 -17508.675} C_VEL
LIN {X 0,Y 295.732,Z 195.455,A -85,B 0,C 180,E1 -17509.236,E2 -17509.236} C_VEL
LIN {X 0,Y 294.464,Z 208.601,A -85,B 0,C 180,E1 -17510.102,E2 -17510.102} C_VEL
LIN {X 0,Y 292.717,Z 220.507,A -85,B 0,C 180,E1 -17511.153,E2 -17511.153} C_VEL
LIN {X 0,Y 290.838,Z 231.251,A -85,B 0,C 180,E1 -17512.4,E2 -17512.4} C_VEL
LIN {X 0,Y 288.599,Z 241.811,A -85,B 0,C 180,E1 -17513.938,E2 -17513.938} C_VEL
LIN {X 0,Y 286.338,Z 251.137,A -85,B 0,C 180,E1 -17515.632,E2 -17515.632} C_VEL
LIN {X 0,Y 284.27,Z 259.247,A -85,B 0,C 180,E1 -17517.472,E2 -17517.472} C_VEL
LIN {X 0,Y 282.087,Z 267.052,A -85,B 0,C 180,E1 -17519.702,E2 -17519.702} C_VEL
LIN {X 0,Y 280.456,Z 272.313,A -85,B 0,C 180,E1 -17521.568,E2 -17521.568} C_VEL
LIN {X 0,Y 278.893,Z 277.343,A -85,B 0,C 180,E1 -17523.833,E2 -17523.833} C_VEL
LIN {X 0,Y 277.693,Z 281.152,A -85,B 0,C 180,E1 -17526.113,E2 -17526.113} C_VEL
LIN {X 0,Y 277.022,Z 283.089,A -85,B 0,C 180,E1 -17527.633,E2 -17527.633} C_VEL
LIN {X 0,Y 276.125,Z 285.375,A -85,B 0,C 180,E1 -17530.347,E2 -17530.347} C_VEL
LIN {X 0,Y 275.701,Z 286.138,A -85,B 0,C 180,E1 -17532.189,E2 -17532.189} C_VEL
LIN {X 0,Y 275.476,Z 286.319,A -85,B 0,C 180,E1 -17533.703,E2 -17533.703} C_VEL
LIN {X 0,Y 275.374,Z 285.809,A -85,B 0,C 180,E1 -17535.891,E2 -17535.891} C_VEL
LIN {X 0,Y 275.395,Z 284.306,A -85,B 0,C 180,E1 -17538.22,E2 -17538.22} C_VEL
LIN {X 0,Y 275.508,Z 282.796,A -85,B 0,C 180,E1 -17539.714,E2 -17539.714} C_VEL
LIN {X 0,Y 275.872,Z 279.711,A -85,B 0,C 180,E1 -17541.946,E2 -17541.946} C_VEL
LIN {X 0,Y 276.357,Z 275.57,A -85,B 0,C 180,E1 -17544.162,E2 -17544.162} C_VEL
LIN {X 0,Y 277.086,Z 269.249,A -85,B 0,C 180,E1 -17546.729,E2 -17546.729} C_VEL
LIN {X 0,Y 277.996,Z 262.373,A -85,B 0,C 180,E1 -17548.914,E2 -17548.914} C_VEL
LIN {X 0,Y 279.013,Z 255.345,A -85,B 0,C 180,E1 -17550.722,E2 -17550.722} C_VEL
LIN {X 0,Y 280.249,Z 246.868,A -85,B 0,C 180,E1 -17552.516,E2 -17552.516} C_VEL
LIN {X 0,Y 281.595,Z 236.41,A -85,B 0,C 180,E1 -17554.294,E2 -17554.294} C_VEL
LIN {X 0,Y 282.905,Z 226.031,A -85,B 0,C 180,E1 -17555.703,E2 -17555.703} C_VEL
LIN {X 0,Y 284.037,Z 214.701,A -85,B 0,C 180,E1 -17556.929,E2 -17556.929} C_VEL
LIN {X 0,Y 284.879,Z 203.122,A -85,B 0,C 180,E1 -17557.888,E2 -17557.888} C_VEL
LIN {X 0,Y 285.609,Z 190.197,A -85,B 0,C 180,E1 -17558.65,E2 -17558.65} C_VEL
LIN {X 0,Y 286.123,Z 176.469,A -85,B 0,C 180,E1 -17559.15,E2 -17559.15} C_VEL
LIN {X 0,Y 287.77,Z 105.749,A -85,B 0,C 180,E1 -17560.898,E2 -17560.898} C_VEL
LIN {X 0,Y 282.713,Z 90.733,A -85,B 0,C 180,E1 -17561.687,E2 -17561.687} C_VEL
LIN {X 0,Y 277.585,Z 78.76,A -85,B 0,C 180,E1 -17562.429,E2 -17562.429} C_VEL
LIN {X 0,Y 277.434,Z 77.933,A -85,B 0,C 180,E1 -17562.482,E2 -17562.482} C_VEL
LIN {X 0,Y 277.411,Z 77.934,A -85,B 0,C 180,E1 -17566.182,E2 -17566.182} C_VEL
LIN {X 0,Y 277.349,Z 77.939,A -85,B 0,C 180,E1 -17570.35,E2 -17570.35} C_VEL
LIN {X 0,Y 277.297,Z 77.945,A -85,B 0,C 180,E1 -17574.158,E2 -17574.158} C_VEL
LIN {X 0,Y 277.328,Z 77.935,A -85,B 0,C 180,E1 -17577.504,E2 -17577.504} C_VEL
LIN {X 0,Y 277.276,Z 77.945,A -85,B 0,C 180,E1 -17580.481,E2 -17580.481} C_VEL
LIN {X 0,Y 277.259,Z 77.943,A -85,B 0,C 180,E1 -17583.895,E2 -17583.895} C_VEL
LIN {X 0,Y 277.286,Z 77.946,A -85,B 0,C 180,E1 -17587.467,E2 -17587.467} C_VEL
LIN {X 0,Y 277.231,Z 77.95,A -85,B 0,C 180,E1 -17591.233,E2 -17591.233} C_VEL
LIN {X 0,Y 277.223,Z 77.951,A -85,B 0,C 180,E1 -17595.222,E2 -17595.222} C_VEL
LIN {X 0,Y 277.226,Z 77.95,A -85,B 0,C 180,E1 -17599.512,E2 -17599.512} C_VEL
LIN {X 0,Y 277.268,Z 77.937,A -85,B 0,C 180,E1 -17602.53,E2 -17602.53} C_VEL
LIN {X 0,Y 277.25,Z 77.935,A -85,B 0,C 180,E1 -17606.104,E2 -17606.104} C_VEL
LIN {X 0,Y 277.265,Z 77.945,A -85,B 0,C 180,E1 -17609.538,E2 -17609.538} C_VEL
LIN {X 0,Y 277.359,Z 77.936,A -85,B 0,C 180,E1 -17612.864,E2 -17612.864} C_VEL
LIN {X 0,Y 277.332,Z 77.932,A -85,B 0,C 180,E1 -17616.079,E2 -17616.079} C_VEL
LIN {X 0,Y 277.348,Z 77.936,A -85,B 0,C 180,E1 -17620.766,E2 -17620.766} C_VEL
LIN {X 0,Y 277.443,Z 77.921,A -85,B 0,C 180,E1 -17624.347,E2 -17624.347} C_VEL
LIN {X 0,Y 276.73,Z 78.011,A -85,B 0,C 180,E1 -17625.558,E2 -17625.558} C_VEL
LIN {X 0,Y 273.841,Z 78.372,A -85,B 0,C 180,E1 -17627.532,E2 -17627.532} C_VEL
LIN {X 0,Y 271.476,Z 78.666,A -85,B 0,C 180,E1 -17629.136,E2 -17629.136} C_VEL
LIN {X 0,Y 270.552,Z 78.78,A -85,B 0,C 180,E1 -17630.379,E2 -17630.379} C_VEL
LIN {X 0,Y 270.524,Z 78.781,A -85,B 0,C 180,E1 -17630.799,E2 -17630.799} C_VEL
LIN {X 0,Y 270.54,Z 78.784,A -85,B 0,C 180,E1 -17634.035,E2 -17634.035} C_VEL
LIN {X 0,Y 270.789,Z 78.75,A -85,B 0,C 180,E1 -17638.512,E2 -17638.512} C_VEL
LIN {X 0,Y 270.789,Z 78.75,A -85,B 0,C 180,E1 -17641.487,E2 -17641.487} C_VEL
LIN {X 0,Y 270.587,Z 78.776,A -85,B 0,C 180,E1 -17647.462,E2 -17647.462} C_VEL
LIN {X 0,Y 270.412,Z 78.798,A -85,B 0,C 180,E1 -17650.482,E2 -17650.482} C_VEL
LIN {X 0,Y 270.405,Z 78.8,A -85,B 0,C 180,E1 -17655.064,E2 -17655.064} C_VEL
LIN {X 0,Y 270.303,Z 78.813,A -85,B 0,C 180,E1 -17659.755,E2 -17659.755} C_VEL
LIN {X 0,Y 270.239,Z 78.822,A -85,B 0,C 180,E1 -17664.589,E2 -17664.589} C_VEL
LIN {X 0,Y 270.274,Z 78.816,A -85,B 0,C 180,E1 -17667.908,E2 -17667.908} C_VEL
LIN {X 0,Y 270.186,Z 78.826,A -85,B 0,C 180,E1 -17671.348,E2 -17671.348} C_VEL
LIN {X 0,Y 270.204,Z 78.827,A -85,B 0,C 180,E1 -17674.905,E2 -17674.905} C_VEL
LIN {X 0,Y 270.199,Z 78.827,A -85,B 0,C 180,E1 -17678.71,E2 -17678.71} C_VEL
LIN {X 0,Y 270.173,Z 78.83,A -85,B 0,C 180,E1 -17682.558,E2 -17682.558} C_VEL
LIN {X 0,Y 270.167,Z 78.831,A -85,B 0,C 180,E1 -17686.751,E2 -17686.751} C_VEL
LIN {X 0,Y 270.224,Z 78.826,A -85,B 0,C 180,E1 -17691.283,E2 -17691.283} C_VEL
LIN {X 0,Y 270.225,Z 78.826,A -85,B 0,C 180,E1 -17695.097,E2 -17695.097} C_VEL
LIN {X 0,Y 270.244,Z 78.994,A -85,B 0,C 180,E1 -17695.816,E2 -17695.816} C_VEL
LIN {X 0,Y 272.629,Z 89.983,A -85,B 0,C 180,E1 -17699.394,E2 -17699.394} C_VEL
LIN {X 0,Y 274.309,Z 98.74,A -85,B 0,C 180,E1 -17702.122,E2 -17702.122} C_VEL
LIN {X 0,Y 274.178,Z 102.416,A -85,B 0,C 180,E1 -17703.185,E2 -17703.185} C_VEL
LIN {X 0,Y 278.873,Z 140.887,A -85,B 0,C 180,E1 -17704.616,E2 -17704.616} C_VEL
LIN {X 0,Y 280.166,Z 153.179,A -85,B 0,C 180,E1 -17705.046,E2 -17705.046} C_VEL
LIN {X 0,Y 278.721,Z 211.423,A -85,B 0,C 180,E1 -17706.551,E2 -17706.551} C_VEL
LIN {X 0,Y 277.89,Z 224.706,A -85,B 0,C 180,E1 -17707.166,E2 -17707.166} C_VEL
LIN {X 0,Y 276.838,Z 236.919,A -85,B 0,C 180,E1 -17708.009,E2 -17708.009} C_VEL
LIN {X 0,Y 275.515,Z 248.406,A -85,B 0,C 180,E1 -17709.076,E2 -17709.076} C_VEL
LIN {X 0,Y 273.952,Z 260.213,A -85,B 0,C 180,E1 -17710.518,E2 -17710.518} C_VEL
LIN {X 0,Y 272.573,Z 270.909,A -85,B 0,C 180,E1 -17712.182,E2 -17712.182} C_VEL
LIN {X 0,Y 271.366,Z 279.51,A -85,B 0,C 180,E1 -17713.834,E2 -17713.834} C_VEL
LIN {X 0,Y 270.296,Z 287.496,A -85,B 0,C 180,E1 -17715.699,E2 -17715.699} C_VEL
LIN {X 0,Y 269.271,Z 295.266,A -85,B 0,C 180,E1 -17717.947,E2 -17717.947} C_VEL
LIN {X 0,Y 268.702,Z 301.509,A -85,B 0,C 180,E1 -17720.211,E2 -17720.211} C_VEL
LIN {X 0,Y 268.402,Z 306.447,A -85,B 0,C 180,E1 -17722.477,E2 -17722.477} C_VEL
LIN {X 0,Y 268.318,Z 309.825,A -85,B 0,C 180,E1 -17724.458,E2 -17724.458} C_VEL
LIN {X 0,Y 268.383,Z 312.958,A -85,B 0,C 180,E1 -17726.997,E2 -17726.997} C_VEL
LIN {X 0,Y 268.413,Z 314.23,A -85,B 0,C 180,E1 -17728.499,E2 -17728.499} C_VEL
LIN {X 0,Y 268.497,Z 315.101,A -85,B 0,C 180,E1 -17729.999,E2 -17729.999} C_VEL
LIN {X 0,Y 268.342,Z 315.52,A -85,B 0,C 180,E1 -17731.5,E2 -17731.5} C_VEL
LIN {X 0,Y 268.315,Z 315.536,A -85,B 0,C 180,E1 -17733.002,E2 -17733.002} C_VEL
LIN {X 0,Y 268.218,Z 314.403,A -85,B 0,C 180,E1 -17736.016,E2 -17736.016} C_VEL
LIN {X 0,Y 268.344,Z 313.238,A -85,B 0,C 180,E1 -17737.524,E2 -17737.524} C_VEL
LIN {X 0,Y 268.801,Z 310.717,A -85,B 0,C 180,E1 -17739.784,E2 -17739.784} C_VEL
LIN {X 0,Y 269.517,Z 307.207,A -85,B 0,C 180,E1 -17742.04,E2 -17742.04} C_VEL
LIN {X 0,Y 270.811,Z 302.644,A -85,B 0,C 180,E1 -17744.272,E2 -17744.272} C_VEL
LIN {X 0,Y 272.424,Z 296.895,A -85,B 0,C 180,E1 -17746.485,E2 -17746.485} C_VEL
LIN {X 0,Y 274.327,Z 289.728,A -85,B 0,C 180,E1 -17748.678,E2 -17748.678} C_VEL
LIN {X 0,Y 276.805,Z 280.871,A -85,B 0,C 180,E1 -17750.821,E2 -17750.821} C_VEL
LIN {X 0,Y 279.507,Z 270.82,A -85,B 0,C 180,E1 -17752.742,E2 -17752.742} C_VEL
LIN {X 0,Y 282.018,Z 260.571,A -85,B 0,C 180,E1 -17754.279,E2 -17754.279} C_VEL
LIN {X 0,Y 284.389,Z 249.248,A -85,B 0,C 180,E1 -17755.624,E2 -17755.624} C_VEL
LIN {X 0,Y 286.553,Z 237.497,A -85,B 0,C 180,E1 -17756.687,E2 -17756.687} C_VEL
LIN {X 0,Y 288.396,Z 224.597,A -85,B 0,C 180,E1 -17757.532,E2 -17757.532} C_VEL
LIN {X 0,Y 289.669,Z 211.05,A -85,B 0,C 180,E1 -17758.13,E2 -17758.13} C_VEL
LIN {X 0,Y 291.681,Z 156.21,A -85,B 0,C 180,E1 -17759.528,E2 -17759.528} C_VEL
LIN {X 0,Y 288.579,Z 135.851,A -85,B 0,C 180,E1 -17760.559,E2 -17760.559} C_VEL
LIN {X 0,Y 285.471,Z 120.573,A -85,B 0,C 180,E1 -17761.471,E2 -17761.471} C_VEL
LIN {X 0,Y 279.951,Z 108.901,A -85,B 0,C 180,E1 -17762.676,E2 -17762.676} C_VEL
LIN {X 0,Y 275.881,Z 100.477,A -85,B 0,C 180,E1 -17763.634,E2 -17763.634} C_VEL
LIN {X 0,Y 273.673,Z 91.094,A -85,B 0,C 180,E1 -17767.242,E2 -17767.242} C_VEL
LIN {X 0,Y 271.34,Z 82.781,A -85,B 0,C 180,E1 -17770.735,E2 -17770.735} C_VEL
LIN {X 0,Y 270.173,Z 78.83,A -85,B 0,C 180,E1 -17772.557,E2 -17772.557} C_VEL
LIN {X 0,Y 270.178,Z 78.816,A -85,B 0,C 180,E1 -17776.747,E2 -17776.747} C_VEL
LIN {X 0,Y 270.211,Z 78.821,A -85,B 0,C 180,E1 -17779.441,E2 -17779.441} C_VEL
LIN {X 0,Y 270.254,Z 78.821,A -85,B 0,C 180,E1 -17783.721,E2 -17783.721} C_VEL
LIN {X 0,Y 270.202,Z 78.825,A -85,B 0,C 180,E1 -17786.893,E2 -17786.893} C_VEL
LIN {X 0,Y 270.226,Z 78.821,A -85,B 0,C 180,E1 -17790.387,E2 -17790.387} C_VEL
LIN {X 0,Y 270.261,Z 78.811,A -85,B 0,C 180,E1 -17793.764,E2 -17793.764} C_VEL
LIN {X 0,Y 270.231,Z 78.812,A -85,B 0,C 180,E1 -17797.039,E2 -17797.039} C_VEL
LIN {X 0,Y 270.3,Z 78.816,A -85,B 0,C 180,E1 -17800.245,E2 -17800.245} C_VEL
LIN {X 0,Y 270.4,Z 78.802,A -85,B 0,C 180,E1 -17804.935,E2 -17804.935} C_VEL
LIN {X 0,Y 270.439,Z 78.797,A -85,B 0,C 180,E1 -17809.519,E2 -17809.519} C_VEL
LIN {X 0,Y 270.605,Z 78.763,A -85,B 0,C 180,E1 -17812.539,E2 -17812.539} C_VEL
LIN {X 0,Y 270.785,Z 78.744,A -85,B 0,C 180,E1 -17818.513,E2 -17818.513} C_VEL
LIN {X 0,Y 270.784,Z 78.748,A -85,B 0,C 180,E1 -17821.488,E2 -17821.488} C_VEL
LIN {X 0,Y 270.582,Z 78.767,A -85,B 0,C 180,E1 -17827.462,E2 -17827.462} C_VEL
LIN {X 0,Y 270.408,Z 78.802,A -85,B 0,C 180,E1 -17830.483,E2 -17830.483} C_VEL
LIN {X 0,Y 270.375,Z 78.807,A -85,B 0,C 180,E1 -17835.067,E2 -17835.067} C_VEL
LIN {X 0,Y 270.259,Z 78.821,A -85,B 0,C 180,E1 -17839.759,E2 -17839.759} C_VEL
LIN {X 0,Y 270.226,Z 78.821,A -85,B 0,C 180,E1 -17844.591,E2 -17844.591} C_VEL
LIN {X 0,Y 270.208,Z 78.828,A -85,B 0,C 180,E1 -17847.916,E2 -17847.916} C_VEL
LIN {X 0,Y 270.172,Z 78.831,A -85,B 0,C 180,E1 -17851.35,E2 -17851.35} C_VEL
LIN {X 0,Y 270.2,Z 78.823,A -85,B 0,C 180,E1 -17854.906,E2 -17854.906} C_VEL
LIN {X 0,Y 270.197,Z 78.832,A -85,B 0,C 180,E1 -17858.711,E2 -17858.711} C_VEL
LIN {X 0,Y 270.166,Z 78.834,A -85,B 0,C 180,E1 -17861.469,E2 -17861.469} C_VEL
LIN {X 0,Y 271.17,Z 81.608,A -85,B 0,C 180,E1 -17861.744,E2 -17861.744} C_VEL
LIN {X 0,Y 273.098,Z 84.234,A -85,B 0,C 180,E1 -17862.172,E2 -17862.172} C_VEL
LIN {X 0,Y 282.065,Z 98.779,A -85,B 0,C 180,E1 -17864.116,E2 -17864.116} C_VEL
LIN {X 0,Y 289.643,Z 113.762,A -85,B 0,C 180,E1 -17865.709,E2 -17865.709} C_VEL
LIN {X 0,Y 293.066,Z 121.307,A -85,B 0,C 180,E1 -17866.411,E2 -17866.411} C_VEL
LIN {X 0,Y 290.732,Z 182.462,A -85,B 0,C 180,E1 -17867.93,E2 -17867.93} C_VEL
LIN {X 0,Y 289.79,Z 195.176,A -85,B 0,C 180,E1 -17868.462,E2 -17868.462} C_VEL
LIN {X 0,Y 288.613,Z 207.268,A -85,B 0,C 180,E1 -17869.25,E2 -17869.25} C_VEL
LIN {X 0,Y 286.959,Z 218.589,A -85,B 0,C 180,E1 -17870.221,E2 -17870.221} C_VEL
LIN {X 0,Y 284.987,Z 229.889,A -85,B 0,C 180,E1 -17871.488,E2 -17871.488} C_VEL
LIN {X 0,Y 282.541,Z 241.122,A -85,B 0,C 180,E1 -17873.105,E2 -17873.105} C_VEL
LIN {X 0,Y 280.223,Z 250.347,A -85,B 0,C 180,E1 -17874.772,E2 -17874.772} C_VEL
LIN {X 0,Y 277.928,Z 258.922,A -85,B 0,C 180,E1 -17876.706,E2 -17876.706} C_VEL
LIN {X 0,Y 275.702,Z 266.7,A -85,B 0,C 180,E1 -17878.923,E2 -17878.923} C_VEL
LIN {X 0,Y 273.939,Z 272.099,A -85,B 0,C 180,E1 -17880.828,E2 -17880.828} C_VEL
LIN {X 0,Y 272.246,Z 277.257,A -85,B 0,C 180,E1 -17883.144,E2 -17883.144} C_VEL
LIN {X 0,Y 270.908,Z 281.188,A -85,B 0,C 180,E1 -17885.476,E2 -17885.476} C_VEL
LIN {X 0,Y 270.168,Z 283.183,A -85,B 0,C 180,E1 -17887.034,E2 -17887.034} C_VEL
LIN {X 0,Y 269.586,Z 284.736,A -85,B 0,C 180,E1 -17888.595,E2 -17888.595} C_VEL
LIN {X 0,Y 269.084,Z 285.805,A -85,B 0,C 180,E1 -17890.152,E2 -17890.152} C_VEL
LIN {X 0,Y 268.708,Z 286.452,A -85,B 0,C 180,E1 -17891.709,E2 -17891.709} C_VEL
LIN {X 0,Y 268.447,Z 286.697,A -85,B 0,C 180,E1 -17893.263,E2 -17893.263} C_VEL
LIN {X 0,Y 268.299,Z 286.201,A -85,B 0,C 180,E1 -17895.746,E2 -17895.746} C_VEL
LIN {X 0,Y 268.289,Z 284.882,A -85,B 0,C 180,E1 -17897.904,E2 -17897.904} C_VEL
LIN {X 0,Y 268.401,Z 283.466,A -85,B 0,C 180,E1 -17899.439,E2 -17899.439} C_VEL
LIN {X 0,Y 268.749,Z 280.485,A -85,B 0,C 180,E1 -17901.731,E2 -17901.731} C_VEL
LIN {X 0,Y 269.213,Z 276.467,A -85,B 0,C 180,E1 -17904.007,E2 -17904.007} C_VEL
LIN {X 0,Y 269.973,Z 270.288,A -85,B 0,C 180,E1 -17906.643,E2 -17906.643} C_VEL
LIN {X 0,Y 270.841,Z 263.563,A -85,B 0,C 180,E1 -17908.885,E2 -17908.885} C_VEL
LIN {X 0,Y 272.127,Z 255.195,A -85,B 0,C 180,E1 -17911.11,E2 -17911.11} C_VEL
LIN {X 0,Y 273.41,Z 246.572,A -85,B 0,C 180,E1 -17912.947,E2 -17912.947} C_VEL
LIN {X 0,Y 274.913,Z 235.6,A -85,B 0,C 180,E1 -17914.822,E2 -17914.822} C_VEL
LIN {X 0,Y 276.169,Z 225.418,A -85,B 0,C 180,E1 -17916.209,E2 -17916.209} C_VEL
LIN {X 0,Y 277.353,Z 213.751,A -85,B 0,C 180,E1 -17917.462,E2 -17917.462} C_VEL
LIN {X 0,Y 278.17,Z 202.974,A -85,B 0,C 180,E1 -17918.354,E2 -17918.354} C_VEL
LIN {X 0,Y 278.922,Z 189.465,A -85,B 0,C 180,E1 -17919.153,E2 -17919.153} C_VEL
LIN {X 0,Y 279.433,Z 175.734,A -85,B 0,C 180,E1 -17919.638,E2 -17919.638} C_VEL
LIN {X 0,Y 281.107,Z 106.936,A -85,B 0,C 180,E1 -17921.374,E2 -17921.374} C_VEL
LIN {X 0,Y 276.108,Z 92.659,A -85,B 0,C 180,E1 -17922.166,E2 -17922.166} C_VEL
LIN {X 0,Y 270.469,Z 79.297,A -85,B 0,C 180,E1 -17923.022,E2 -17923.022} C_VEL
LIN {X 0,Y 270.391,Z 78.809,A -85,B 0,C 180,E1 -17923.044,E2 -17923.044} C_VEL
LIN {X 0,Y 270.36,Z 78.811,A -85,B 0,C 180,E1 -17926.616,E2 -17926.616} C_VEL
LIN {X 0,Y 270.296,Z 78.816,A -85,B 0,C 180,E1 -17930.601,E2 -17930.601} C_VEL
LIN {X 0,Y 270.242,Z 78.822,A -85,B 0,C 180,E1 -17934.589,E2 -17934.589} C_VEL
LIN {X 0,Y 270.274,Z 78.814,A -85,B 0,C 180,E1 -17937.909,E2 -17937.909} C_VEL
LIN {X 0,Y 270.188,Z 78.828,A -85,B 0,C 180,E1 -17941.348,E2 -17941.348} C_VEL
LIN {X 0,Y 270.219,Z 78.818,A -85,B 0,C 180,E1 -17944.903,E2 -17944.903} C_VEL
LIN {X 0,Y 270.226,Z 78.822,A -85,B 0,C 180,E1 -17948.717,E2 -17948.717} C_VEL
LIN {X 0,Y 270.196,Z 78.826,A -85,B 0,C 180,E1 -17952.554,E2 -17952.554} C_VEL
LIN {X 0,Y 270.175,Z 78.827,A -85,B 0,C 180,E1 -17956.749,E2 -17956.749} C_VEL
LIN {X 0,Y 270.201,Z 78.819,A -85,B 0,C 180,E1 -17961.289,E2 -17961.289} C_VEL
LIN {X 0,Y 270.205,Z 78.808,A -85,B 0,C 180,E1 -17965.094,E2 -17965.094} C_VEL
LIN {X 0,Y 270.204,Z 78.826,A -85,B 0,C 180,E1 -17969.13,E2 -17969.13} C_VEL
LIN {X 0,Y 270.266,Z 78.818,A -85,B 0,C 180,E1 -17972.146,E2 -17972.146} C_VEL
LIN {X 0,Y 270.28,Z 78.809,A -85,B 0,C 180,E1 -17975.519,E2 -17975.519} C_VEL
LIN {X 0,Y 270.305,Z 78.815,A -85,B 0,C 180,E1 -17980.244,E2 -17980.244} C_VEL
LIN {X 0,Y 270.406,Z 78.798,A -85,B 0,C 180,E1 -17984.935,E2 -17984.935} C_VEL
LIN {X 0,Y 270.416,Z 78.798,A -85,B 0,C 180,E1 -17989.518,E2 -17989.518} C_VEL
LIN {X 0,Y 270.524,Z 78.781,A -85,B 0,C 180,E1 -17990.799,E2 -17990.799} C_VEL
LIN {X 0,Y 269.964,Z 78.855,A -85,B 0,C 180,E1 -17992.04,E2 -17992.04} C_VEL
LIN {X 0,Y 267.103,Z 79.216,A -85,B 0,C 180,E1 -17994.061,E2 -17994.061} C_VEL
LIN {X 0,Y 264.646,Z 79.52,A -85,B 0,C 180,E1 -17995.706,E2 -17995.706} C_VEL
LIN {X 0,Y 263.649,Z 79.641,A -85,B 0,C 180,E1 -17996.982,E2 -17996.982} C_VEL
LIN {X 0,Y 263.603,Z 79.644,A -85,B 0,C 180,E1 -17997.414,E2 -17997.414} C_VEL
LIN {X 0,Y 263.805,Z 79.619,A -85,B 0,C 180,E1 -18000,E2 -18000} C_VEL
LIN {X 0,Y 263.564,Z 79.652,A -85,B 0,C 180,E1 -18003.057,E2 -18003.057} C_VEL
LIN {X 0,Y 263.546,Z 79.652,A -85,B 0,C 180,E1 -18007.662,E2 -18007.662} C_VEL
LIN {X 0,Y 263.352,Z 79.678,A -85,B 0,C 180,E1 -18010.766,E2 -18010.766} C_VEL
LIN {X 0,Y 263.353,Z 79.676,A -85,B 0,C 180,E1 -18015.478,E2 -18015.478} C_VEL
LIN {X 0,Y 263.265,Z 79.689,A -85,B 0,C 180,E1 -18020.306,E2 -18020.306} C_VEL
LIN {X 0,Y 263.194,Z 79.698,A -85,B 0,C 180,E1 -18025.293,E2 -18025.293} C_VEL
LIN {X 0,Y 263.181,Z 79.7,A -85,B 0,C 180,E1 -18028.729,E2 -18028.729} C_VEL
LIN {X 0,Y 263.135,Z 79.705,A -85,B 0,C 180,E1 -18032.288,E2 -18032.288} C_VEL
LIN {X 0,Y 263.184,Z 79.702,A -85,B 0,C 180,E1 -18036.763,E2 -18036.763} C_VEL
LIN {X 0,Y 263.126,Z 79.708,A -85,B 0,C 180,E1 -18041.593,E2 -18041.593} C_VEL
LIN {X 0,Y 263.124,Z 79.706,A -85,B 0,C 180,E1 -18046.016,E2 -18046.016} C_VEL
LIN {X 0,Y 263.117,Z 79.712,A -85,B 0,C 180,E1 -18050.129,E2 -18050.129} C_VEL
LIN {X 0,Y 263.191,Z 79.704,A -85,B 0,C 180,E1 -18054.022,E2 -18054.022} C_VEL
LIN {X 0,Y 263.219,Z 79.887,A -85,B 0,C 180,E1 -18055.375,E2 -18055.375} C_VEL
LIN {X 0,Y 265.803,Z 91.924,A -85,B 0,C 180,E1 -18059.403,E2 -18059.403} C_VEL
LIN {X 0,Y 267.397,Z 100.518,A -85,B 0,C 180,E1 -18062.148,E2 -18062.148} C_VEL
LIN {X 0,Y 267.413,Z 102.252,A -85,B 0,C 180,E1 -18062.61,E2 -18062.61} C_VEL
LIN {X 0,Y 271.886,Z 138.663,A -85,B 0,C 180,E1 -18064.014,E2 -18064.014} C_VEL
LIN {X 0,Y 273.473,Z 153.823,A -85,B 0,C 180,E1 -18064.56,E2 -18064.56} C_VEL
LIN {X 0,Y 271.983,Z 211.416,A -85,B 0,C 180,E1 -18066.086,E2 -18066.086} C_VEL
LIN {X 0,Y 271.086,Z 225.349,A -85,B 0,C 180,E1 -18066.762,E2 -18066.762} C_VEL
LIN {X 0,Y 269.88,Z 238.342,A -85,B 0,C 180,E1 -18067.714,E2 -18067.714} C_VEL
LIN {X 0,Y 268.457,Z 250.171,A -85,B 0,C 180,E1 -18068.901,E2 -18068.901} C_VEL
LIN {X 0,Y 266.799,Z 261.564,A -85,B 0,C 180,E1 -18070.375,E2 -18070.375} C_VEL
LIN {X 0,Y 265.415,Z 272.16,A -85,B 0,C 180,E1 -18072.131,E2 -18072.131} C_VEL
LIN {X 0,Y 264.295,Z 280.289,A -85,B 0,C 180,E1 -18073.786,E2 -18073.786} C_VEL
LIN {X 0,Y 263.029,Z 289.432,A -85,B 0,C 180,E1 -18076.085,E2 -18076.085} C_VEL
LIN {X 0,Y 262.021,Z 296.775,A -85,B 0,C 180,E1 -18078.394,E2 -18078.394} C_VEL
LIN {X 0,Y 261.536,Z 302.65,A -85,B 0,C 180,E1 -18080.721,E2 -18080.721} C_VEL
LIN {X 0,Y 261.298,Z 307.252,A -85,B 0,C 180,E1 -18083.048,E2 -18083.048} C_VEL
LIN {X 0,Y 261.233,Z 310.729,A -85,B 0,C 180,E1 -18085.37,E2 -18085.37} C_VEL
LIN {X 0,Y 261.308,Z 312.453,A -85,B 0,C 180,E1 -18086.916,E2 -18086.916} C_VEL
LIN {X 0,Y 261.331,Z 313.752,A -85,B 0,C 180,E1 -18088.458,E2 -18088.458} C_VEL
LIN {X 0,Y 261.408,Z 314.65,A -85,B 0,C 180,E1 -18089.999,E2 -18089.999} C_VEL
LIN {X 0,Y 261.262,Z 315.12,A -85,B 0,C 180,E1 -18091.541,E2 -18091.541} C_VEL
LIN {X 0,Y 261.24,Z 315.164,A -85,B 0,C 180,E1 -18093.084,E2 -18093.084} C_VEL
LIN {X 0,Y 261.143,Z 314.082,A -85,B 0,C 180,E1 -18096.179,E2 -18096.179} C_VEL
LIN {X 0,Y 261.29,Z 312.963,A -85,B 0,C 180,E1 -18097.728,E2 -18097.728} C_VEL
LIN {X 0,Y 261.583,Z 311.401,A -85,B 0,C 180,E1 -18099.276,E2 -18099.276} C_VEL
LIN {X 0,Y 262.242,Z 308.293,A -85,B 0,C 180,E1 -18101.595,E2 -18101.595} C_VEL
LIN {X 0,Y 263.418,Z 304.161,A -85,B 0,C 180,E1 -18103.893,E2 -18103.893} C_VEL
LIN {X 0,Y 265.299,Z 297.876,A -85,B 0,C 180,E1 -18106.545,E2 -18106.545} C_VEL
LIN {X 0,Y 267.197,Z 291.201,A -85,B 0,C 180,E1 -18108.756,E2 -18108.756} C_VEL
LIN {X 0,Y 269.721,Z 282.672,A -85,B 0,C 180,E1 -18110.994,E2 -18110.994} C_VEL
LIN {X 0,Y 272.226,Z 274.048,A -85,B 0,C 180,E1 -18112.783,E2 -18112.783} C_VEL
LIN {X 0,Y 274.921,Z 263.47,A -85,B 0,C 180,E1 -18114.544,E2 -18114.544} C_VEL
LIN {X 0,Y 277.416,Z 252.994,A -85,B 0,C 180,E1 -18115.912,E2 -18115.912} C_VEL
LIN {X 0,Y 279.745,Z 241.446,A -85,B 0,C 180,E1 -18117.087,E2 -18117.087} C_VEL
LIN {X 0,Y 281.858,Z 228.208,A -85,B 0,C 180,E1 -18118.075,E2 -18118.075} C_VEL
LIN {X 0,Y 283.393,Z 215.275,A -85,B 0,C 180,E1 -18118.74,E2 -18118.74} C_VEL
LIN {X 0,Y 284.22,Z 200.864,A -85,B 0,C 180,E1 -18119.194,E2 -18119.194} C_VEL
LIN {X 0,Y 285.748,Z 156.724,A -85,B 0,C 180,E1 -18120.322,E2 -18120.322} C_VEL
LIN {X 0,Y 282.791,Z 137.291,A -85,B 0,C 180,E1 -18121.345,E2 -18121.345} C_VEL
LIN {X 0,Y 280.074,Z 123.716,A -85,B 0,C 180,E1 -18122.183,E2 -18122.183} C_VEL
LIN {X 0,Y 273.329,Z 109.337,A -85,B 0,C 180,E1 -18123.732,E2 -18123.732} C_VEL
LIN {X 0,Y 268.589,Z 99.939,A -85,B 0,C 180,E1 -18124.91,E2 -18124.91} C_VEL
LIN {X 0,Y 266.845,Z 92.756,A -85,B 0,C 180,E1 -18127.803,E2 -18127.803} C_VEL
LIN {X 0,Y 264.882,Z 85.638,A -85,B 0,C 180,E1 -18130.873,E2 -18130.873} C_VEL
LIN {X 0,Y 263.107,Z 79.706,A -85,B 0,C 180,E1 -18133.715,E2 -18133.715} C_VEL
LIN {X 0,Y 263.145,Z 79.707,A -85,B 0,C 180,E1 -18138.111,E2 -18138.111} C_VEL
LIN {X 0,Y 263.186,Z 79.694,A -85,B 0,C 180,E1 -18142.108,E2 -18142.108} C_VEL
LIN {X 0,Y 263.181,Z 79.694,A -85,B 0,C 180,E1 -18145.89,E2 -18145.89} C_VEL
LIN {X 0,Y 263.148,Z 79.698,A -85,B 0,C 180,E1 -18149.507,E2 -18149.507} C_VEL
LIN {X 0,Y 263.19,Z 79.691,A -85,B 0,C 180,E1 -18153.003,E2 -18153.003} C_VEL
LIN {X 0,Y 263.182,Z 79.695,A -85,B 0,C 180,E1 -18156.387,E2 -18156.387} C_VEL
LIN {X 0,Y 263.262,Z 79.691,A -85,B 0,C 180,E1 -18159.693,E2 -18159.693} C_VEL
LIN {X 0,Y 263.349,Z 79.683,A -85,B 0,C 180,E1 -18164.522,E2 -18164.522} C_VEL
LIN {X 0,Y 263.372,Z 79.677,A -85,B 0,C 180,E1 -18169.235,E2 -18169.235} C_VEL
LIN {X 0,Y 263.567,Z 79.639,A -85,B 0,C 180,E1 -18172.339,E2 -18172.339} C_VEL
LIN {X 0,Y 263.749,Z 79.62,A -85,B 0,C 180,E1 -18178.473,E2 -18178.473} C_VEL
LIN {X 0,Y 263.748,Z 79.624,A -85,B 0,C 180,E1 -18181.527,E2 -18181.527} C_VEL
LIN {X 0,Y 263.542,Z 79.643,A -85,B 0,C 180,E1 -18187.663,E2 -18187.663} C_VEL
LIN {X 0,Y 263.347,Z 79.682,A -85,B 0,C 180,E1 -18190.767,E2 -18190.767} C_VEL
LIN {X 0,Y 263.322,Z 79.685,A -85,B 0,C 180,E1 -18195.48,E2 -18195.48} C_VEL
LIN {X 0,Y 263.237,Z 79.695,A -85,B 0,C 180,E1 -18200.309,E2 -18200.309} C_VEL
LIN {X 0,Y 263.171,Z 79.695,A -85,B 0,C 180,E1 -18205.296,E2 -18205.296} C_VEL
LIN {X 0,Y 263.137,Z 79.701,A -85,B 0,C 180,E1 -18208.735,E2 -18208.735} C_VEL
LIN {X 0,Y 263.127,Z 79.703,A -85,B 0,C 180,E1 -18212.29,E2 -18212.29} C_VEL
LIN {X 0,Y 263.18,Z 79.705,A -85,B 0,C 180,E1 -18216.763,E2 -18216.763} C_VEL
LIN {X 0,Y 263.113,Z 79.714,A -85,B 0,C 180,E1 -18220.184,E2 -18220.184} C_VEL
LIN {X 0,Y 264.166,Z 82.602,A -85,B 0,C 180,E1 -18220.491,E2 -18220.491} C_VEL
LIN {X 0,Y 266.016,Z 84.951,A -85,B 0,C 180,E1 -18220.924,E2 -18220.924} C_VEL
LIN {X 0,Y 268.247,Z 88.326,A -85,B 0,C 180,E1 -18221.452,E2 -18221.452} C_VEL
LIN {X 0,Y 277.435,Z 103.356,A -85,B 0,C 180,E1 -18223.529,E2 -18223.529} C_VEL
LIN {X 0,Y 284.477,Z 117.419,A -85,B 0,C 180,E1 -18225.069,E2 -18225.069} C_VEL
LIN {X 0,Y 287.177,Z 123.362,A -85,B 0,C 180,E1 -18225.649,E2 -18225.649} C_VEL
LIN {X 0,Y 284.733,Z 184.201,A -85,B 0,C 180,E1 -18227.197,E2 -18227.197} C_VEL
LIN {X 0,Y 283.651,Z 197.257,A -85,B 0,C 180,E1 -18227.788,E2 -18227.788} C_VEL
LIN {X 0,Y 282.36,Z 209.713,A -85,B 0,C 180,E1 -18228.656,E2 -18228.656} C_VEL
LIN {X 0,Y 280.661,Z 220.321,A -85,B 0,C 180,E1 -18229.615,E2 -18229.615} C_VEL
LIN {X 0,Y 278.373,Z 232.328,A -85,B 0,C 180,E1 -18231.043,E2 -18231.043} C_VEL
LIN {X 0,Y 275.79,Z 243.529,A -85,B 0,C 180,E1 -18232.756,E2 -18232.756} C_VEL
LIN {X 0,Y 273.194,Z 253.187,A -85,B 0,C 180,E1 -18234.633,E2 -18234.633} C_VEL
LIN {X 0,Y 271.078,Z 260.53,A -85,B 0,C 180,E1 -18236.408,E2 -18236.408} C_VEL
LIN {X 0,Y 268.964,Z 267.507,A -85,B 0,C 180,E1 -18238.494,E2 -18238.494} C_VEL
LIN {X 0,Y 266.762,Z 273.88,A -85,B 0,C 180,E1 -18240.888,E2 -18240.888} C_VEL
LIN {X 0,Y 265.079,Z 278.639,A -85,B 0,C 180,E1 -18243.211,E2 -18243.211} C_VEL
LIN {X 0,Y 263.748,Z 282.314,A -85,B 0,C 180,E1 -18245.606,E2 -18245.606} C_VEL
LIN {X 0,Y 262.715,Z 284.893,A -85,B 0,C 180,E1 -18248.006,E2 -18248.006} C_VEL
LIN {X 0,Y 262.102,Z 286.164,A -85,B 0,C 180,E1 -18249.802,E2 -18249.802} C_VEL
LIN {X 0,Y 261.431,Z 287.065,A -85,B 0,C 180,E1 -18252.8,E2 -18252.8} C_VEL
LIN {X 0,Y 261.203,Z 286.588,A -85,B 0,C 180,E1 -18255.613,E2 -18255.613} C_VEL
LIN {X 0,Y 261.203,Z 285.458,A -85,B 0,C 180,E1 -18257.57,E2 -18257.57} C_VEL
LIN {X 0,Y 261.271,Z 284.098,A -85,B 0,C 180,E1 -18259.147,E2 -18259.147} C_VEL
LIN {X 0,Y 261.602,Z 281.225,A -85,B 0,C 180,E1 -18261.504,E2 -18261.504} C_VEL
LIN {X 0,Y 262.085,Z 277.319,A -85,B 0,C 180,E1 -18263.843,E2 -18263.843} C_VEL
LIN {X 0,Y 262.69,Z 272.289,A -85,B 0,C 180,E1 -18266.165,E2 -18266.165} C_VEL
LIN {X 0,Y 263.52,Z 265.978,A -85,B 0,C 180,E1 -18268.472,E2 -18268.472} C_VEL
LIN {X 0,Y 264.76,Z 258.045,A -85,B 0,C 180,E1 -18270.761,E2 -18270.761} C_VEL
LIN {X 0,Y 266.021,Z 249.961,A -85,B 0,C 180,E1 -18272.65,E2 -18272.65} C_VEL
LIN {X 0,Y 267.472,Z 240.106,A -85,B 0,C 180,E1 -18274.522,E2 -18274.522} C_VEL
LIN {X 0,Y 268.949,Z 229.06,A -85,B 0,C 180,E1 -18276.189,E2 -18276.189} C_VEL
LIN {X 0,Y 270.146,Z 218.262,A -85,B 0,C 180,E1 -18277.475,E2 -18277.475} C_VEL
LIN {X 0,Y 271.236,Z 205.298,A -85,B 0,C 180,E1 -18278.663,E2 -18278.663} C_VEL
LIN {X 0,Y 272.103,Z 192.654,A -85,B 0,C 180,E1 -18279.478,E2 -18279.478} C_VEL
LIN {X 0,Y 272.663,Z 179.436,A -85,B 0,C 180,E1 -18280.02,E2 -18280.02} C_VEL
LIN {X 0,Y 274.458,Z 108.314,A -85,B 0,C 180,E1 -18281.867,E2 -18281.867} C_VEL
LIN {X 0,Y 269.626,Z 94.731,A -85,B 0,C 180,E1 -18282.656,E2 -18282.656} C_VEL
LIN {X 0,Y 263.385,Z 80.112,A -85,B 0,C 180,E1 -18283.637,E2 -18283.637} C_VEL
LIN {X 0,Y 263.338,Z 79.688,A -85,B 0,C 180,E1 -18283.738,E2 -18283.738} C_VEL
LIN {X 0,Y 263.276,Z 79.692,A -85,B 0,C 180,E1 -18287.076,E2 -18287.076} C_VEL
LIN {X 0,Y 263.219,Z 79.696,A -85,B 0,C 180,E1 -18290.849,E2 -18290.849} C_VEL
LIN {X 0,Y 263.197,Z 79.699,A -85,B 0,C 180,E1 -18295.293,E2 -18295.293} C_VEL
LIN {X 0,Y 263.17,Z 79.7,A -85,B 0,C 180,E1 -18298.731,E2 -18298.731} C_VEL
LIN {X 0,Y 263.138,Z 79.702,A -85,B 0,C 180,E1 -18302.288,E2 -18302.288} C_VEL
LIN {X 0,Y 263.193,Z 79.7,A -85,B 0,C 180,E1 -18305.978,E2 -18305.978} C_VEL
LIN {X 0,Y 263.127,Z 79.706,A -85,B 0,C 180,E1 -18309.869,E2 -18309.869} C_VEL
LIN {X 0,Y 263.137,Z 79.703,A -85,B 0,C 180,E1 -18313.982,E2 -18313.982} C_VEL
LIN {X 0,Y 263.129,Z 79.706,A -85,B 0,C 180,E1 -18318.406,E2 -18318.406} C_VEL
LIN {X 0,Y 263.185,Z 79.681,A -85,B 0,C 180,E1 -18323.237,E2 -18323.237} C_VEL
LIN {X 0,Y 263.136,Z 79.699,A -85,B 0,C 180,E1 -18327.712,E2 -18327.712} C_VEL
LIN {X 0,Y 263.199,Z 79.698,A -85,B 0,C 180,E1 -18331.785,E2 -18331.785} C_VEL
LIN {X 0,Y 263.229,Z 79.688,A -85,B 0,C 180,E1 -18335.2,E2 -18335.2} C_VEL
LIN {X 0,Y 263.267,Z 79.689,A -85,B 0,C 180,E1 -18339.693,E2 -18339.693} C_VEL
LIN {X 0,Y 263.354,Z 79.676,A -85,B 0,C 180,E1 -18344.522,E2 -18344.522} C_VEL
LIN {X 0,Y 263.358,Z 79.677,A -85,B 0,C 180,E1 -18349.233,E2 -18349.233} C_VEL
LIN {X 0,Y 263.561,Z 79.65,A -85,B 0,C 180,E1 -18352.338,E2 -18352.338} C_VEL
LIN {X 0,Y 263.603,Z 79.644,A -85,B 0,C 180,E1 -18357.414,E2 -18357.414} C_VEL
LIN {X 0,Y 263.355,Z 79.676,A -85,B 0,C 180,E1 -18358.269,E2 -18358.269} C_VEL
LIN {X 0,Y 262.05,Z 79.839,A -85,B 0,C 180,E1 -18359.53,E2 -18359.53} C_VEL
LIN {X 0,Y 257.623,Z 80.391,A -85,B 0,C 180,E1 -18362.463,E2 -18362.463} C_VEL
LIN {X 0,Y 256.483,Z 80.538,A -85,B 0,C 180,E1 -18363.777,E2 -18363.777} C_VEL
LIN {X 0,Y 256.365,Z 80.546,A -85,B 0,C 180,E1 -18364.223,E2 -18364.223} C_VEL
LIN {X 0,Y 256.506,Z 80.527,A -85,B 0,C 180,E1 -18367.874,E2 -18367.874} C_VEL
LIN {X 0,Y 256.287,Z 80.559,A -85,B 0,C 180,E1 -18372.672,E2 -18372.672} C_VEL
LIN {X 0,Y 256.285,Z 80.555,A -85,B 0,C 180,E1 -18376.302,E2 -18376.302} C_VEL
LIN {X 0,Y 256.156,Z 80.577,A -85,B 0,C 180,E1 -18381.117,E2 -18381.117} C_VEL
LIN {X 0,Y 256.172,Z 80.574,A -85,B 0,C 180,E1 -18385.129,E2 -18385.129} C_VEL
LIN {X 0,Y 256.116,Z 80.575,A -85,B 0,C 180,E1 -18389.599,E2 -18389.599} C_VEL
LIN {X 0,Y 256.069,Z 80.586,A -85,B 0,C 180,E1 -18393.292,E2 -18393.292} C_VEL
LIN {X 0,Y 256.116,Z 80.58,A -85,B 0,C 180,E1 -18397.27,E2 -18397.27} C_VEL
LIN {X 0,Y 256.056,Z 80.588,A -85,B 0,C 180,E1 -18401.203,E2 -18401.203} C_VEL
LIN {X 0,Y 256.059,Z 80.583,A -85,B 0,C 180,E1 -18405.53,E2 -18405.53} C_VEL
LIN {X 0,Y 256.058,Z 80.59,A -85,B 0,C 180,E1 -18408.797,E2 -18408.797} C_VEL
LIN {X 0,Y 256.146,Z 80.58,A -85,B 0,C 180,E1 -18412.87,E2 -18412.87} C_VEL
LIN {X 0,Y 256.158,Z 80.694,A -85,B 0,C 180,E1 -18414.875,E2 -18414.875} C_VEL
LIN {X 0,Y 258.661,Z 92.388,A -85,B 0,C 180,E1 -18418.919,E2 -18418.919} C_VEL
LIN {X 0,Y 260.423,Z 101.561,A -85,B 0,C 180,E1 -18421.943,E2 -18421.943} C_VEL
LIN {X 0,Y 261.894,Z 110.947,A -85,B 0,C 180,E1 -18422.375,E2 -18422.375} C_VEL
LIN {X 0,Y 266.677,Z 152.229,A -85,B 0,C 180,E1 -18423.978,E2 -18423.978} C_VEL
LIN {X 0,Y 266.132,Z 183.032,A -85,B 0,C 180,E1 -18424.812,E2 -18424.812} C_VEL
LIN {X 0,Y 265.287,Z 211.289,A -85,B 0,C 180,E1 -18425.599,E2 -18425.599} C_VEL
LIN {X 0,Y 264.338,Z 225.134,A -85,B 0,C 180,E1 -18426.288,E2 -18426.288} C_VEL
LIN {X 0,Y 263.175,Z 237.575,A -85,B 0,C 180,E1 -18427.218,E2 -18427.218} C_VEL
LIN {X 0,Y 261.592,Z 250.286,A -85,B 0,C 180,E1 -18428.527,E2 -18428.527} C_VEL
LIN {X 0,Y 259.888,Z 261.591,A -85,B 0,C 180,E1 -18430.037,E2 -18430.037} C_VEL
LIN {X 0,Y 258.435,Z 272.189,A -85,B 0,C 180,E1 -18431.857,E2 -18431.857} C_VEL
LIN {X 0,Y 257.188,Z 281.157,A -85,B 0,C 180,E1 -18433.772,E2 -18433.772} C_VEL
LIN {X 0,Y 255.885,Z 289.958,A -85,B 0,C 180,E1 -18436.094,E2 -18436.094} C_VEL
LIN {X 0,Y 254.908,Z 297.108,A -85,B 0,C 180,E1 -18438.469,E2 -18438.469} C_VEL
LIN {X 0,Y 254.38,Z 303.639,A -85,B 0,C 180,E1 -18441.259,E2 -18441.259} C_VEL
LIN {X 0,Y 254.159,Z 307.917,A -85,B 0,C 180,E1 -18443.649,E2 -18443.649} C_VEL
LIN {X 0,Y 254.147,Z 310.177,A -85,B 0,C 180,E1 -18445.241,E2 -18445.241} C_VEL
LIN {X 0,Y 254.234,Z 311.948,A -85,B 0,C 180,E1 -18446.83,E2 -18446.83} C_VEL
LIN {X 0,Y 254.251,Z 313.274,A -85,B 0,C 180,E1 -18448.415,E2 -18448.415} C_VEL
LIN {X 0,Y 254.321,Z 314.198,A -85,B 0,C 180,E1 -18449.999,E2 -18449.999} C_VEL
LIN {X 0,Y 254.185,Z 314.709,A -85,B 0,C 180,E1 -18451.584,E2 -18451.584} C_VEL
LIN {X 0,Y 254.143,Z 314.79,A -85,B 0,C 180,E1 -18453.17,E2 -18453.17} C_VEL
LIN {X 0,Y 254.085,Z 314.294,A -85,B 0,C 180,E1 -18455.279,E2 -18455.279} C_VEL
LIN {X 0,Y 254.231,Z 312.677,A -85,B 0,C 180,E1 -18457.944,E2 -18457.944} C_VEL
LIN {X 0,Y 254.545,Z 311.167,A -85,B 0,C 180,E1 -18459.535,E2 -18459.535} C_VEL
LIN {X 0,Y 255.25,Z 308.117,A -85,B 0,C 180,E1 -18461.917,E2 -18461.917} C_VEL
LIN {X 0,Y 256.497,Z 304.046,A -85,B 0,C 180,E1 -18464.276,E2 -18464.276} C_VEL
LIN {X 0,Y 258.469,Z 297.837,A -85,B 0,C 180,E1 -18466.995,E2 -18466.995} C_VEL
LIN {X 0,Y 260.292,Z 291.796,A -85,B 0,C 180,E1 -18469.088,E2 -18469.088} C_VEL
LIN {X 0,Y 262.622,Z 284.304,A -85,B 0,C 180,E1 -18471.178,E2 -18471.178} C_VEL
LIN {X 0,Y 265.161,Z 276.129,A -85,B 0,C 180,E1 -18473.013,E2 -18473.013} C_VEL
LIN {X 0,Y 267.899,Z 266.195,A -85,B 0,C 180,E1 -18474.818,E2 -18474.818} C_VEL
LIN {X 0,Y 270.745,Z 255.011,A -85,B 0,C 180,E1 -18476.393,E2 -18476.393} C_VEL
LIN {X 0,Y 273.117,Z 244.094,A -85,B 0,C 180,E1 -18477.592,E2 -18477.592} C_VEL
LIN {X 0,Y 275.314,Z 232.045,A -85,B 0,C 180,E1 -18478.596,E2 -18478.596} C_VEL
LIN {X 0,Y 277.07,Z 219.06,A -85,B 0,C 180,E1 -18479.366,E2 -18479.366} C_VEL
LIN {X 0,Y 278.181,Z 205.316,A -85,B 0,C 180,E1 -18479.884,E2 -18479.884} C_VEL
LIN {X 0,Y 279.976,Z 158.079,A -85,B 0,C 180,E1 -18481.111,E2 -18481.111} C_VEL
LIN {X 0,Y 277.179,Z 139.214,A -85,B 0,C 180,E1 -18482.135,E2 -18482.135} C_VEL
LIN {X 0,Y 274.645,Z 126.489,A -85,B 0,C 180,E1 -18482.95,E2 -18482.95} C_VEL
LIN {X 0,Y 267.534,Z 111.64,A -85,B 0,C 180,E1 -18484.65,E2 -18484.65} C_VEL
LIN {X 0,Y 263.222,Z 103.472,A -85,B 0,C 180,E1 -18485.724,E2 -18485.724} C_VEL
LIN {X 0,Y 261.305,Z 99.422,A -85,B 0,C 180,E1 -18486.277,E2 -18486.277} C_VEL
LIN {X 0,Y 259.075,Z 90.77,A -85,B 0,C 180,E1 -18489.984,E2 -18489.984} C_VEL
LIN {X 0,Y 256.798,Z 83.154,A -85,B 0,C 180,E1 -18493.589,E2 -18493.589} C_VEL
LIN {X 0,Y 256.057,Z 80.569,A -85,B 0,C 180,E1 -18494.918,E2 -18494.918} C_VEL
LIN {X 0,Y 256.083,Z 80.582,A -85,B 0,C 180,E1 -18498.802,E2 -18498.802} C_VEL
LIN {X 0,Y 256.152,Z 80.57,A -85,B 0,C 180,E1 -18502.871,E2 -18502.871} C_VEL
LIN {X 0,Y 256.083,Z 80.583,A -85,B 0,C 180,E1 -18506.71,E2 -18506.71} C_VEL
LIN {X 0,Y 256.136,Z 80.58,A -85,B 0,C 180,E1 -18511.404,E2 -18511.404} C_VEL
LIN {X 0,Y 256.165,Z 80.575,A -85,B 0,C 180,E1 -18515.699,E2 -18515.699} C_VEL
LIN {X 0,Y 256.165,Z 80.572,A -85,B 0,C 180,E1 -18519.105,E2 -18519.105} C_VEL
LIN {X 0,Y 256.298,Z 80.557,A -85,B 0,C 180,E1 -18524.085,E2 -18524.085} C_VEL
LIN {X 0,Y 256.308,Z 80.555,A -85,B 0,C 180,E1 -18528.934,E2 -18528.934} C_VEL
LIN {X 0,Y 256.535,Z 80.515,A -85,B 0,C 180,E1 -18532.127,E2 -18532.127} C_VEL
LIN {X 0,Y 256.712,Z 80.495,A -85,B 0,C 180,E1 -18538.432,E2 -18538.432} C_VEL
LIN {X 0,Y 256.711,Z 80.5,A -85,B 0,C 180,E1 -18541.569,E2 -18541.569} C_VEL
LIN {X 0,Y 256.461,Z 80.531,A -85,B 0,C 180,E1 -18546.715,E2 -18546.715} C_VEL
LIN {X 0,Y 256.425,Z 80.537,A -85,B 0,C 180,E1 -18549.465,E2 -18549.465} C_VEL
LIN {X 0,Y 256.235,Z 80.562,A -85,B 0,C 180,E1 -18554.292,E2 -18554.292} C_VEL
LIN {X 0,Y 256.176,Z 80.562,A -85,B 0,C 180,E1 -18557.565,E2 -18557.565} C_VEL
LIN {X 0,Y 256.14,Z 80.57,A -85,B 0,C 180,E1 -18561.111,E2 -18561.111} C_VEL
LIN {X 0,Y 256.158,Z 80.569,A -85,B 0,C 180,E1 -18565.125,E2 -18565.125} C_VEL
LIN {X 0,Y 256.056,Z 80.582,A -85,B 0,C 180,E1 -18569.608,E2 -18569.608} C_VEL
LIN {X 0,Y 256.065,Z 80.586,A -85,B 0,C 180,E1 -18573.294,E2 -18573.294} C_VEL
LIN {X 0,Y 256.112,Z 80.582,A -85,B 0,C 180,E1 -18577.271,E2 -18577.271} C_VEL
LIN {X 0,Y 256.12,Z 80.776,A -85,B 0,C 180,E1 -18578.819,E2 -18578.819} C_VEL
LIN {X 0,Y 257.006,Z 83.332,A -85,B 0,C 180,E1 -18579.099,E2 -18579.099} C_VEL
LIN {X 0,Y 259.087,Z 85.91,A -85,B 0,C 180,E1 -18579.619,E2 -18579.619} C_VEL
LIN {X 0,Y 261.477,Z 89.458,A -85,B 0,C 180,E1 -18580.222,E2 -18580.222} C_VEL
LIN {X 0,Y 271.124,Z 104.892,A -85,B 0,C 180,E1 -18582.53,E2 -18582.53} C_VEL
LIN {X 0,Y 277.125,Z 116.413,A -85,B 0,C 180,E1 -18583.904,E2 -18583.904} C_VEL
LIN {X 0,Y 281.417,Z 125.771,A -85,B 0,C 180,E1 -18584.872,E2 -18584.872} C_VEL
LIN {X 0,Y 278.886,Z 184.494,A -85,B 0,C 180,E1 -18586.38,E2 -18586.38} C_VEL
LIN {X 0,Y 277.731,Z 198.058,A -85,B 0,C 180,E1 -18587.011,E2 -18587.011} C_VEL
LIN {X 0,Y 276.337,Z 210.584,A -85,B 0,C 180,E1 -18587.906,E2 -18587.906} C_VEL
LIN {X 0,Y 274.409,Z 222.012,A -85,B 0,C 180,E1 -18588.983,E2 -18588.983} C_VEL
LIN {X 0,Y 272.04,Z 233.692,A -85,B 0,C 180,E1 -18590.434,E2 -18590.434} C_VEL
LIN {X 0,Y 269.624,Z 243.619,A -85,B 0,C 180,E1 -18591.99,E2 -18591.99} C_VEL
LIN {X 0,Y 267.15,Z 252.47,A -85,B 0,C 180,E1 -18593.708,E2 -18593.708} C_VEL
LIN {X 0,Y 264.627,Z 260.867,A -85,B 0,C 180,E1 -18595.752,E2 -18595.752} C_VEL
LIN {X 0,Y 262.231,Z 268.314,A -85,B 0,C 180,E1 -18598.041,E2 -18598.041} C_VEL
LIN {X 0,Y 260.168,Z 273.991,A -85,B 0,C 180,E1 -18600.227,E2 -18600.227} C_VEL
LIN {X 0,Y 258.457,Z 278.565,A -85,B 0,C 180,E1 -18602.467,E2 -18602.467} C_VEL
LIN {X 0,Y 257.313,Z 281.584,A -85,B 0,C 180,E1 -18604.335,E2 -18604.335} C_VEL
LIN {X 0,Y 255.867,Z 285.05,A -85,B 0,C 180,E1 -18607.385,E2 -18607.385} C_VEL
LIN {X 0,Y 255.098,Z 286.561,A -85,B 0,C 180,E1 -18609.508,E2 -18609.508} C_VEL
LIN {X 0,Y 254.414,Z 287.434,A -85,B 0,C 180,E1 -18612.311,E2 -18612.311} C_VEL
LIN {X 0,Y 254.113,Z 286.975,A -85,B 0,C 180,E1 -18615.467,E2 -18615.467} C_VEL
LIN {X 0,Y 254.109,Z 286.031,A -85,B 0,C 180,E1 -18617.218,E2 -18617.218} C_VEL
LIN {X 0,Y 254.149,Z 284.723,A -85,B 0,C 180,E1 -18618.839,E2 -18618.839} C_VEL
LIN {X 0,Y 254.463,Z 281.956,A -85,B 0,C 180,E1 -18621.263,E2 -18621.263} C_VEL
LIN {X 0,Y 254.938,Z 278.164,A -85,B 0,C 180,E1 -18623.67,E2 -18623.67} C_VEL
LIN {X 0,Y 255.562,Z 273.251,A -85,B 0,C 180,E1 -18626.058,E2 -18626.058} C_VEL
LIN {X 0,Y 256.402,Z 267.074,A -85,B 0,C 180,E1 -18628.43,E2 -18628.43} C_VEL
LIN {X 0,Y 257.646,Z 259.369,A -85,B 0,C 180,E1 -18630.782,E2 -18630.782} C_VEL
LIN {X 0,Y 259.21,Z 249.684,A -85,B 0,C 180,E1 -18633.109,E2 -18633.109} C_VEL
LIN {X 0,Y 260.71,Z 239.698,A -85,B 0,C 180,E1 -18635.027,E2 -18635.027} C_VEL
LIN {X 0,Y 262.233,Z 228.729,A -85,B 0,C 180,E1 -18636.688,E2 -18636.688} C_VEL
LIN {X 0,Y 263.502,Z 217.351,A -85,B 0,C 180,E1 -18638.05,E2 -18638.05} C_VEL
LIN {X 0,Y 264.556,Z 205.141,A -85,B 0,C 180,E1 -18639.172,E2 -18639.172} C_VEL
LIN {X 0,Y 265.424,Z 192.203,A -85,B 0,C 180,E1 -18640.007,E2 -18640.007} C_VEL
LIN {X 0,Y 266.022,Z 178.444,A -85,B 0,C 180,E1 -18640.561,E2 -18640.561} C_VEL
LIN {X 0,Y 267.944,Z 110.145,A -85,B 0,C 180,E1 -18642.36,E2 -18642.36} C_VEL
LIN {X 0,Y 263.599,Z 97.865,A -85,B 0,C 180,E1 -18643.097,E2 -18643.097} C_VEL
LIN {X 0,Y 256.418,Z 81.296,A -85,B 0,C 180,E1 -18644.261,E2 -18644.261} C_VEL
LIN {X 0,Y 256.276,Z 80.569,A -85,B 0,C 180,E1 -18644.34,E2 -18644.34} C_VEL
LIN {X 0,Y 256.216,Z 80.572,A -85,B 0,C 180,E1 -18647.562,E2 -18647.562} C_VEL
LIN {X 0,Y 256.158,Z 80.575,A -85,B 0,C 180,E1 -18651.118,E2 -18651.118} C_VEL
LIN {X 0,Y 256.175,Z 80.574,A -85,B 0,C 180,E1 -18655.13,E2 -18655.13} C_VEL
LIN {X 0,Y 256.108,Z 80.582,A -85,B 0,C 180,E1 -18659.601,E2 -18659.601} C_VEL
LIN {X 0,Y 256.089,Z 80.578,A -85,B 0,C 180,E1 -18663.29,E2 -18663.29} C_VEL
LIN {X 0,Y 256.133,Z 80.579,A -85,B 0,C 180,E1 -18667.275,E2 -18667.275} C_VEL
LIN {X 0,Y 256.079,Z 80.584,A -85,B 0,C 180,E1 -18671.199,E2 -18671.199} C_VEL
LIN {X 0,Y 256.07,Z 80.583,A -85,B 0,C 180,E1 -18674.472,E2 -18674.472} C_VEL
LIN {X 0,Y 256.059,Z 80.588,A -85,B 0,C 180,E1 -18678.797,E2 -18678.797} C_VEL
LIN {X 0,Y 256.133,Z 80.561,A -85,B 0,C 180,E1 -18682.867,E2 -18682.867} C_VEL
LIN {X 0,Y 256.071,Z 80.572,A -85,B 0,C 180,E1 -18686.707,E2 -18686.707} C_VEL
LIN {X 0,Y 256.107,Z 80.581,A -85,B 0,C 180,E1 -18690.399,E2 -18690.399} C_VEL
LIN {X 0,Y 256.192,Z 80.566,A -85,B 0,C 180,E1 -18694.861,E2 -18694.861} C_VEL
LIN {X 0,Y 256.171,Z 80.574,A -85,B 0,C 180,E1 -18699.105,E2 -18699.105} C_VEL
LIN {X 0,Y 256.303,Z 80.552,A -85,B 0,C 180,E1 -18704.085,E2 -18704.085} C_VEL
LIN {X 0,Y 256.301,Z 80.556,A -85,B 0,C 180,E1 -18708.933,E2 -18708.933} C_VEL
LIN {X 0,Y 256.518,Z 80.526,A -85,B 0,C 180,E1 -18712.126,E2 -18712.126} C_VEL
LIN {X 0,Y 256.559,Z 80.52,A -85,B 0,C 180,E1 -18717.457,E2 -18717.457} C_VEL
LIN {X 0,Y 256.768,Z 80.495,A -85,B 0,C 180,E1 -18720,E2 -18720} C_VEL
LIN {X 0,Y 256.499,Z 80.532,A -85,B 0,C 180,E1 -18723.141,E2 -18723.141} C_VEL
LIN {X 0,Y 256.365,Z 80.546,A -85,B 0,C 180,E1 -18724.223,E2 -18724.223} C_VEL
LIN {X 0,Y 255.63,Z 80.643,A -85,B 0,C 180,E1 -18725.535,E2 -18725.535} C_VEL
LIN {X 0,Y 252.756,Z 80.995,A -85,B 0,C 180,E1 -18727.675,E2 -18727.675} C_VEL
LIN {X 0,Y 250.355,Z 81.296,A -85,B 0,C 180,E1 -18729.417,E2 -18729.417} C_VEL
LIN {X 0,Y 249.327,Z 81.426,A -85,B 0,C 180,E1 -18730.767,E2 -18730.767} C_VEL
LIN {X 0,Y 249.242,Z 81.438,A -85,B 0,C 180,E1 -18731.224,E2 -18731.224} C_VEL
LIN {X 0,Y 249.208,Z 81.439,A -85,B 0,C 180,E1 -18734.703,E2 -18734.703} C_VEL
LIN {X 0,Y 249.142,Z 81.449,A -85,B 0,C 180,E1 -18738.077,E2 -18738.077} C_VEL
LIN {X 0,Y 249.086,Z 81.456,A -85,B 0,C 180,E1 -18741.518,E2 -18741.518} C_VEL
LIN {X 0,Y 249.119,Z 81.451,A -85,B 0,C 180,E1 -18745.475,E2 -18745.475} C_VEL
LIN {X 0,Y 249.085,Z 81.453,A -85,B 0,C 180,E1 -18748.993,E2 -18748.993} C_VEL
LIN {X 0,Y 249.032,Z 81.462,A -85,B 0,C 180,E1 -18752.425,E2 -18752.425} C_VEL
LIN {X 0,Y 249.05,Z 81.464,A -85,B 0,C 180,E1 -18756.342,E2 -18756.342} C_VEL
LIN {X 0,Y 249.007,Z 81.467,A -85,B 0,C 180,E1 -18760.478,E2 -18760.478} C_VEL
LIN {X 0,Y 249.004,Z 81.46,A -85,B 0,C 180,E1 -18764.879,E2 -18764.879} C_VEL
LIN {X 0,Y 249.018,Z 81.466,A -85,B 0,C 180,E1 -18767.362,E2 -18767.362} C_VEL
LIN {X 0,Y 249.04,Z 81.466,A -85,B 0,C 180,E1 -18771.621,E2 -18771.621} C_VEL
LIN {X 0,Y 249.108,Z 81.492,A -85,B 0,C 180,E1 -18774.351,E2 -18774.351} C_VEL
LIN {X 0,Y 251.518,Z 92.835,A -85,B 0,C 180,E1 -18778.404,E2 -18778.404} C_VEL
LIN {X 0,Y 253.242,Z 101.272,A -85,B 0,C 180,E1 -18781.275,E2 -18781.275} C_VEL
LIN {X 0,Y 254.731,Z 107.186,A -85,B 0,C 180,E1 -18781.598,E2 -18781.598} C_VEL
LIN {X 0,Y 259.71,Z 149.588,A -85,B 0,C 180,E1 -18783.319,E2 -18783.319} C_VEL
LIN {X 0,Y 260.149,Z 155.929,A -85,B 0,C 180,E1 -18783.543,E2 -18783.543} C_VEL
LIN {X 0,Y 258.599,Z 211.141,A -85,B 0,C 180,E1 -18785.086,E2 -18785.086} C_VEL
LIN {X 0,Y 257.615,Z 224.906,A -85,B 0,C 180,E1 -18785.79,E2 -18785.79} C_VEL
LIN {X 0,Y 256.363,Z 237.801,A -85,B 0,C 180,E1 -18786.791,E2 -18786.791} C_VEL
LIN {X 0,Y 254.736,Z 250.386,A -85,B 0,C 180,E1 -18788.132,E2 -18788.132} C_VEL
LIN {X 0,Y 252.987,Z 261.596,A -85,B 0,C 180,E1 -18789.68,E2 -18789.68} C_VEL
LIN {X 0,Y 251.733,Z 270.715,A -85,B 0,C 180,E1 -18791.272,E2 -18791.272} C_VEL
LIN {X 0,Y 250.367,Z 279.117,A -85,B 0,C 180,E1 -18793.048,E2 -18793.048} C_VEL
LIN {X 0,Y 249.125,Z 287.715,A -85,B 0,C 180,E1 -18795.291,E2 -18795.291} C_VEL
LIN {X 0,Y 248.021,Z 295.23,A -85,B 0,C 180,E1 -18797.729,E2 -18797.729} C_VEL
LIN {X 0,Y 247.434,Z 301.264,A -85,B 0,C 180,E1 -18800.187,E2 -18800.187} C_VEL
LIN {X 0,Y 247.146,Z 306.01,A -85,B 0,C 180,E1 -18802.647,E2 -18802.647} C_VEL
LIN {X 0,Y 247.06,Z 309.606,A -85,B 0,C 180,E1 -18805.104,E2 -18805.104} C_VEL
LIN {X 0,Y 247.138,Z 311.436,A -85,B 0,C 180,E1 -18806.739,E2 -18806.739} C_VEL
LIN {X 0,Y 247.173,Z 312.792,A -85,B 0,C 180,E1 -18808.37,E2 -18808.37} C_VEL
LIN {X 0,Y 247.237,Z 313.743,A -85,B 0,C 180,E1 -18809.999,E2 -18809.999} C_VEL
LIN {X 0,Y 247.109,Z 314.284,A -85,B 0,C 180,E1 -18811.629,E2 -18811.629} C_VEL
LIN {X 0,Y 247.051,Z 314.417,A -85,B 0,C 180,E1 -18813.261,E2 -18813.261} C_VEL
LIN {X 0,Y 246.989,Z 314.029,A -85,B 0,C 180,E1 -18815.181,E2 -18815.181} C_VEL
LIN {X 0,Y 247.171,Z 312.386,A -85,B 0,C 180,E1 -18818.173,E2 -18818.173} C_VEL
LIN {X 0,Y 247.523,Z 310.93,A -85,B 0,C 180,E1 -18819.808,E2 -18819.808} C_VEL
LIN {X 0,Y 248.274,Z 307.926,A -85,B 0,C 180,E1 -18822.257,E2 -18822.257} C_VEL
LIN {X 0,Y 249.596,Z 303.912,A -85,B 0,C 180,E1 -18824.679,E2 -18824.679} C_VEL
LIN {X 0,Y 251.669,Z 297.798,A -85,B 0,C 180,E1 -18827.469,E2 -18827.469} C_VEL
LIN {X 0,Y 253.795,Z 291.154,A -85,B 0,C 180,E1 -18829.829,E2 -18829.829} C_VEL
LIN {X 0,Y 256.506,Z 282.951,A -85,B 0,C 180,E1 -18832.131,E2 -18832.131} C_VEL
LIN {X 0,Y 259.215,Z 274.592,A -85,B 0,C 180,E1 -18833.996,E2 -18833.996} C_VEL
LIN {X 0,Y 262.113,Z 264.345,A -85,B 0,C 180,E1 -18835.83,E2 -18835.83} C_VEL
LIN {X 0,Y 265.128,Z 252.81,A -85,B 0,C 180,E1 -18837.424,E2 -18837.424} C_VEL
LIN {X 0,Y 267.651,Z 241.46,A -85,B 0,C 180,E1 -18838.633,E2 -18838.633} C_VEL
LIN {X 0,Y 269.727,Z 229.814,A -85,B 0,C 180,E1 -18839.566,E2 -18839.566} C_VEL
LIN {X 0,Y 271.512,Z 216.355,A -85,B 0,C 180,E1 -18840.321,E2 -18840.321} C_VEL
LIN {X 0,Y 272.465,Z 204.109,A -85,B 0,C 180,E1 -18840.763,E2 -18840.763} C_VEL
LIN {X 0,Y 274.166,Z 158.808,A -85,B 0,C 180,E1 -18841.971,E2 -18841.971} C_VEL
LIN {X 0,Y 271.335,Z 139.575,A -85,B 0,C 180,E1 -18843.056,E2 -18843.056} C_VEL
LIN {X 0,Y 269.308,Z 129.562,A -85,B 0,C 180,E1 -18843.729,E2 -18843.729} C_VEL
LIN {X 0,Y 261.518,Z 113.089,A -85,B 0,C 180,E1 -18845.699,E2 -18845.699} C_VEL
LIN {X 0,Y 256.008,Z 102.897,A -85,B 0,C 180,E1 -18847.152,E2 -18847.152} C_VEL
LIN {X 0,Y 254.006,Z 98.88,A -85,B 0,C 180,E1 -18847.759,E2 -18847.759} C_VEL
LIN {X 0,Y 251.984,Z 91.433,A -85,B 0,C 180,E1 -18851.145,E2 -18851.145} C_VEL
LIN {X 0,Y 249.502,Z 83.282,A -85,B 0,C 180,E1 -18855.235,E2 -18855.235} C_VEL
LIN {X 0,Y 249.021,Z 81.444,A -85,B 0,C 180,E1 -18856.24,E2 -18856.24} C_VEL
LIN {X 0,Y 249.036,Z 81.458,A -85,B 0,C 180,E1 -18859.636,E2 -18859.636} C_VEL
LIN {X 0,Y 249.072,Z 81.458,A -85,B 0,C 180,E1 -18863.662,E2 -18863.662} C_VEL
LIN {X 0,Y 249.038,Z 81.464,A -85,B 0,C 180,E1 -18867.844,E2 -18867.844} C_VEL
LIN {X 0,Y 249.095,Z 81.457,A -85,B 0,C 180,E1 -18871.338,E2 -18871.338} C_VEL
LIN {X 0,Y 249.149,Z 81.449,A -85,B 0,C 180,E1 -18874.969,E2 -18874.969} C_VEL
LIN {X 0,Y 249.11,Z 81.455,A -85,B 0,C 180,E1 -18880.212,E2 -18880.212} C_VEL
LIN {X 0,Y 249.24,Z 81.433,A -85,B 0,C 180,E1 -18883.622,E2 -18883.622} C_VEL
LIN {X 0,Y 249.251,Z 81.429,A -85,B 0,C 180,E1 -18888.617,E2 -18888.617} C_VEL
LIN {X 0,Y 249.477,Z 81.395,A -85,B 0,C 180,E1 -18891.903,E2 -18891.903} C_VEL
LIN {X 0,Y 249.432,Z 81.403,A -85,B 0,C 180,E1 -18896.77,E2 -18896.77} C_VEL
LIN {X 0,Y 249.726,Z 81.379,A -85,B 0,C 180,E1 -18900,E2 -18900} C_VEL
LIN {X 0,Y 249.43,Z 81.399,A -85,B 0,C 180,E1 -18903.231,E2 -18903.231} C_VEL
LIN {X 0,Y 249.432,Z 81.408,A -85,B 0,C 180,E1 -18906.699,E2 -18906.699} C_VEL
LIN {X 0,Y 249.34,Z 81.422,A -85,B 0,C 180,E1 -18909.737,E2 -18909.737} C_VEL
LIN {X 0,Y 249.181,Z 81.444,A -85,B 0,C 180,E1 -18914.705,E2 -18914.705} C_VEL
LIN {X 0,Y 249.111,Z 81.443,A -85,B 0,C 180,E1 -18918.08,E2 -18918.08} C_VEL
LIN {X 0,Y 249.079,Z 81.447,A -85,B 0,C 180,E1 -18921.519,E2 -18921.519} C_VEL
LIN {X 0,Y 249.103,Z 81.446,A -85,B 0,C 180,E1 -18925.47,E2 -18925.47} C_VEL
LIN {X 0,Y 249.04,Z 81.456,A -85,B 0,C 180,E1 -18928.977,E2 -18928.977} C_VEL
LIN {X 0,Y 249.026,Z 81.459,A -85,B 0,C 180,E1 -18932.427,E2 -18932.427} C_VEL
LIN {X 0,Y 249.102,Z 81.456,A -85,B 0,C 180,E1 -18937.163,E2 -18937.163} C_VEL
LIN {X 0,Y 249.103,Z 81.73,A -85,B 0,C 180,E1 -18937.329,E2 -18937.329} C_VEL
LIN {X 0,Y 250.106,Z 84.38,A -85,B 0,C 180,E1 -18937.661,E2 -18937.661} C_VEL
LIN {X 0,Y 252.111,Z 86.753,A -85,B 0,C 180,E1 -18938.197,E2 -18938.197} C_VEL
LIN {X 0,Y 254.377,Z 90.245,A -85,B 0,C 180,E1 -18938.816,E2 -18938.816} C_VEL
LIN {X 0,Y 261.985,Z 101.812,A -85,B 0,C 180,E1 -18940.767,E2 -18940.767} C_VEL
LIN {X 0,Y 269.013,Z 113.822,A -85,B 0,C 180,E1 -18942.468,E2 -18942.468} C_VEL
LIN {X 0,Y 275.649,Z 127.953,A -85,B 0,C 180,E1 -18944.044,E2 -18944.044} C_VEL
LIN {X 0,Y 273.125,Z 184.525,A -85,B 0,C 180,E1 -18945.521,E2 -18945.521} C_VEL
LIN {X 0,Y 271.966,Z 197.754,A -85,B 0,C 180,E1 -18946.132,E2 -18946.132} C_VEL
LIN {X 0,Y 270.455,Z 210.783,A -85,B 0,C 180,E1 -18947.067,E2 -18947.067} C_VEL
LIN {X 0,Y 268.515,Z 222.002,A -85,B 0,C 180,E1 -18948.132,E2 -18948.132} C_VEL
LIN {X 0,Y 266.267,Z 232.748,A -85,B 0,C 180,E1 -18949.463,E2 -18949.463} C_VEL
LIN {X 0,Y 263.508,Z 243.739,A -85,B 0,C 180,E1 -18951.189,E2 -18951.189} C_VEL
LIN {X 0,Y 260.656,Z 253.527,A -85,B 0,C 180,E1 -18953.137,E2 -18953.137} C_VEL
LIN {X 0,Y 258.145,Z 261.448,A -85,B 0,C 180,E1 -18955.13,E2 -18955.13} C_VEL
LIN {X 0,Y 255.525,Z 269.128,A -85,B 0,C 180,E1 -18957.567,E2 -18957.567} C_VEL
LIN {X 0,Y 253.2,Z 275.213,A -85,B 0,C 180,E1 -18960.026,E2 -18960.026} C_VEL
LIN {X 0,Y 251.308,Z 279.945,A -85,B 0,C 180,E1 -18962.521,E2 -18962.521} C_VEL
LIN {X 0,Y 249.828,Z 283.48,A -85,B 0,C 180,E1 -18965.042,E2 -18965.042} C_VEL
LIN {X 0,Y 249.037,Z 285.208,A -85,B 0,C 180,E1 -18966.729,E2 -18966.729} C_VEL
LIN {X 0,Y 248.12,Z 286.952,A -85,B 0,C 180,E1 -18969.186,E2 -18969.186} C_VEL
LIN {X 0,Y 247.412,Z 287.803,A -85,B 0,C 180,E1 -18971.793,E2 -18971.793} C_VEL
LIN {X 0,Y 247.154,Z 287.804,A -85,B 0,C 180,E1 -18973.48,E2 -18973.48} C_VEL
LIN {X 0,Y 247.044,Z 287.365,A -85,B 0,C 180,E1 -18975.297,E2 -18975.297} C_VEL
LIN {X 0,Y 247.001,Z 286.604,A -85,B 0,C 180,E1 -18976.843,E2 -18976.843} C_VEL
LIN {X 0,Y 247.033,Z 285.348,A -85,B 0,C 180,E1 -18978.514,E2 -18978.514} C_VEL
LIN {X 0,Y 247.325,Z 282.687,A -85,B 0,C 180,E1 -18981.009,E2 -18981.009} C_VEL
LIN {X 0,Y 247.819,Z 279.004,A -85,B 0,C 180,E1 -18983.487,E2 -18983.487} C_VEL
LIN {X 0,Y 248.438,Z 274.211,A -85,B 0,C 180,E1 -18985.945,E2 -18985.945} C_VEL
LIN {X 0,Y 249.289,Z 268.165,A -85,B 0,C 180,E1 -18988.385,E2 -18988.385} C_VEL
LIN {X 0,Y 250.531,Z 260.632,A -85,B 0,C 180,E1 -18990.804,E2 -18990.804} C_VEL
LIN {X 0,Y 251.833,Z 252.938,A -85,B 0,C 180,E1 -18992.8,E2 -18992.8} C_VEL
